RoboDK station: kr30 cnc 070119 curve 7 axis test 3.rdk

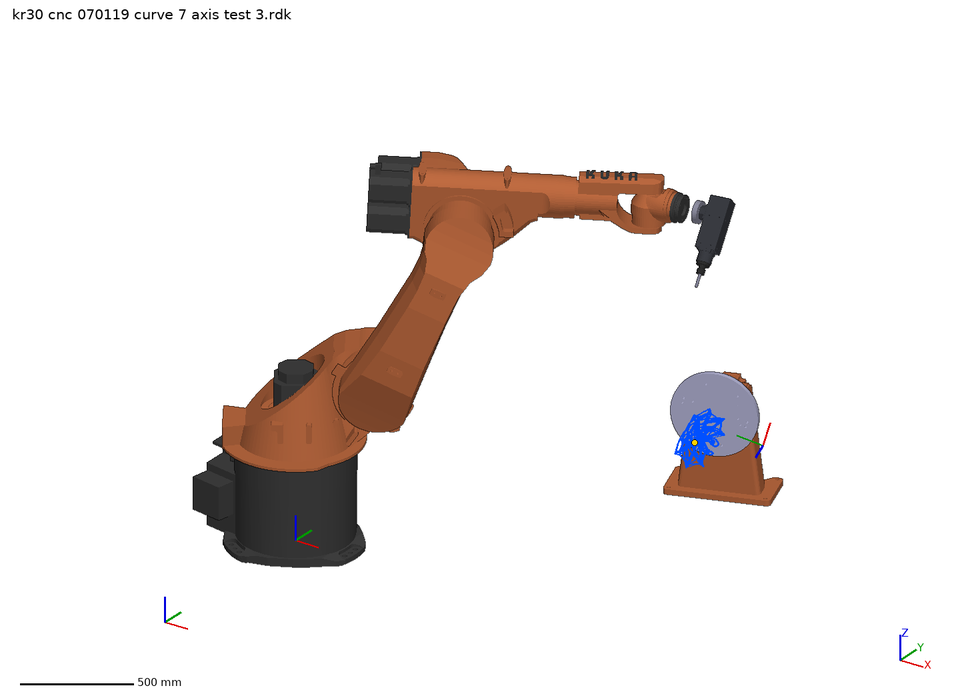
[picture v0: the station drawn from its stored meshes, robots at their saved joint values, targets as dots, program paths as lines]
Station kr30 cnc 070119 curve 7 axis test 3. Poses are relative to the parent item; angles as X-Y-Z fixed-axis rotations.
  - machining project Curve settings: C:/Temp/temp3/RhinoProject.stl | rotZ(0) | rotX(0)*rotY(0) | rotz(0) | onStart | onPathStart | onApproach | onPoint | onRetract | onFinish | onPathFinish | M_RunCode(%1)
  - frame KUKA KP1 MD250 Base at (0, 1000, 0) mm
    - robot KUKA KP1 MD250: 1 axes, payload 250 kg
        modified DH rows (alpha deg, a mm, theta deg, d mm): 0, 0, 0, 0
        base shift (1750, 1710, 820) mm, rotated rx 0 ry 90 rz -70 deg
        joint limits [-3600] to [3600]; home [0]; saved at [883.939]
      - frame Reference Rhino at (0, -260, 100) mm
        - object RhinoPart at (0, 0, 0) mm
  - frame KUKA KR 30 HA Base at (0, 2000, 0) mm
    - robot KUKA KR 30 HA: 6 axes, payload 30 kg, reach 2033 mm, repeatability 0.05 mm, weight 665 kg
        modified DH rows (alpha deg, a mm, theta deg, d mm): 0, 0, 0, 815; -90, 350, 0, 0; 0, 850, -90, 0; -90, 145, 0, 820; 90, 0, 0, 0; -90, 0, 180, 170
        joint limits [-185, -135, -120, -350, -119, -350] to [185, 35, 158, 350, 119, 350]; home [0, -90, 90, 0, 0, 0]; saved at [-33.388, -63.686, 66.526, 94.328, 22.372, -52.483]
      - tool 1/2" End Mill TCP, TCP at (337.71, -2.2, 160.57) mm, rotated rx 0 ry 90 rz 0 deg, size 415.8 x 102 x 153.6 mm
  - machining project RhinoPart Settings: rotZ(0) | rotX(0)*rotY(-65) | rotz(50) | onStart | onPathStart | onApproach | onPoint | onRetract | onFinish | onPathFinish | M_RunCode(%1)
  - program RhinoPart (1342 instructions, listed below)
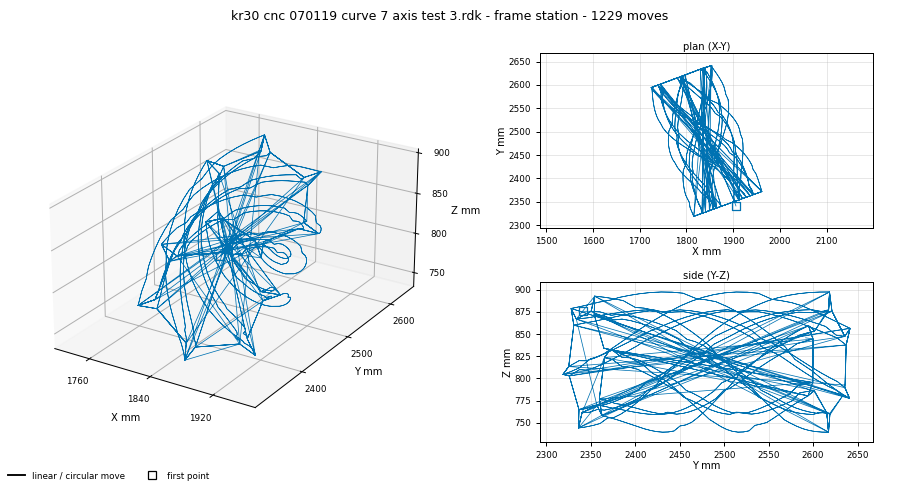
[picture p0: tool path of kr30 cnc 070119 curve 7 axis test 3.rdk in frame station, 1229 of 1229 moves have a stored position in this frame; points joined in program order, loops and branches not executed]

--- program RhinoPart (robot KUKA KR 30 HA) ---
  Set Ref.: Reference Rhino
  Set Tool: 1/2" End Mill TCP
  Show 1/2" End Mill TCP
  Set speed (1000.0 mm/s)
  MoveJ 1 to (58.93, 255.88, 300) mm, rotated rx 180 ry -65 rz 136 deg; joints [2.666, 0.348, 23.749, -54.366, 106.166, -75.82, 24.002]
  MoveL 2 to (58.93, 255.88, 300) mm, rotated rx 180 ry -65 rz 136 deg; joints [2.666, 0.348, 23.749, -54.366, 106.166, -75.82, 24.002]
  MoveL 3 to (58.93, 255.88, 290) mm, rotated rx 180 ry -65 rz 136 deg; joints [2.402, -0.635, 25.77, -54.277, 105.366, -75.09, 24.002]
  MoveL 4 to (58.93, 255.88, 290) mm, rotated rx 180 ry -65 rz 136 deg; joints [2.402, -0.635, 25.77, -54.277, 105.366, -75.09, 24.002]
  Set speed (60.0 mm/s)
  MoveL 5 to (37.11, 300.24, 290) mm, rotated rx -180 ry -65 rz -172.69 deg; joints [2.418, -1.215, 26.671, -54.196, 105.19, -74.811, -27.315]
  MoveL 6 to (-37.11, 208.63, 290) mm, rotated rx -180 ry -65 rz 14.16 deg; joints [2.386, -0.033, 24.818, -54.365, 105.558, -75.393, 145.844]
  Set speed (60.0 mm/s)
  MoveL 7 to (-58.93, 252.99, 290) mm, rotated rx -180 ry -65 rz -33.22 deg; joints [2.401, -0.598, 25.711, -54.282, 105.378, -75.109, 193.216]
  MoveL 8 to (21.11, 199.39, 290) mm, rotated rx -180 ry -65 rz 69.21 deg; joints [2.383, 0.084, 24.632, -54.382, 105.596, -75.453, 90.794]
  Set speed (60.0 mm/s)
  MoveL 9 to (34.79, 183.72, 290) mm, rotated rx -180 ry -65 rz 74.51 deg; joints [2.31, 3.521, 18.897, -54.969, 106.871, -77.447, 85.485]
  MoveL 10 to (21.11, 199.39, 290) mm, rotated rx -180 ry -65 rz 69.21 deg; joints [2.383, 0.084, 24.632, -54.382, 105.596, -75.453, 90.794]
  Set speed (60.0 mm/s)
  MoveL 11 to (-28.22, 202.67, 290) mm, rotated rx 180 ry -65 rz 23.79 deg; joints [2.384, 0.043, 24.698, -54.376, 105.583, -75.432, 136.207]
  MoveL 12 to (-43.85, 188.95, 290) mm, rotated rx 180 ry -65 rz 18.32 deg; joints [2.311, 3.444, 19.031, -54.954, 106.839, -77.397, 141.679]
  Set speed (60.0 mm/s)
  MoveL 13 to (-28.22, 202.67, 290) mm, rotated rx -180 ry -65 rz 23.79 deg; joints [2.384, 0.043, 24.698, -54.376, 105.583, -75.432, 136.207]
  MoveL 14 to (-43.85, 188.95, 290) mm, rotated rx 180 ry -65 rz 18.32 deg; joints [2.311, 3.444, 19.031, -54.954, 106.839, -77.397, 141.679]
  Set speed (60.0 mm/s)
  MoveL 15 to (-37.11, 208.63, 290) mm, rotated rx -180 ry -65 rz 14.16 deg; joints [2.386, -0.033, 24.818, -54.365, 105.558, -75.393, 145.844]
  MoveL 16 to (-78.63, 259.66, 290) mm, rotated rx 180 ry -65 rz -39.75 deg; joints [2.329, 2.455, 20.731, -54.77, 106.443, -76.78, 199.755]
  Set speed (60.0 mm/s)
  MoveL 17 to (-58.93, 252.99, 290) mm, rotated rx -180 ry -65 rz -33.22 deg; joints [2.401, -0.598, 25.711, -54.282, 105.378, -75.109, 193.216]
  MoveL 18 to (-78.63, 259.66, 290) mm, rotated rx -180 ry -65 rz -39.75 deg; joints [2.329, 2.455, 20.731, -54.77, 106.443, -76.78, 199.755]
  Set speed (60.0 mm/s)
  MoveL 19 to (-58.22, 263.67, 290) mm, rotated rx -180 ry -65 rz -43.61 deg; joints [2.405, -0.736, 25.927, -54.263, 105.335, -75.041, 203.606]
  MoveL 20 to (-30.72, 304.75, 290) mm, rotated rx -180 ry -65 rz -95.53 deg; joints [2.42, -1.275, 26.764, -54.188, 105.172, -74.782, 255.533]
  Set speed (60.0 mm/s)
  MoveL 21 to (-58.22, 263.67, 290) mm, rotated rx -180 ry -65 rz -43.61 deg; joints [2.405, -0.736, 25.927, -54.263, 105.335, -75.041, 203.606]
  MoveL 22 to (-30.72, 304.75, 290) mm, rotated rx -180 ry -65 rz -95.53 deg; joints [2.42, -1.275, 26.764, -54.188, 105.172, -74.782, 255.533]
  Set speed (60.0 mm/s)
  MoveL 23 to (-34.79, 325.15, 290) mm, rotated rx 180 ry -65 rz -101.9 deg; joints [2.347, 1.599, 22.168, -54.622, 106.121, -76.277, 261.899]
  MoveL 24 to (-21.11, 309.47, 290) mm, rotated rx -180 ry -65 rz -106.89 deg; joints [2.421, -1.338, 26.861, -54.18, 105.153, -74.752, 266.89]
  Set speed (60.0 mm/s)
  MoveL 25 to (-34.79, 325.15, 290) mm, rotated rx -180 ry -65 rz -101.9 deg; joints [2.347, 1.599, 22.168, -54.622, 106.121, -76.277, 261.899]
  MoveL 26 to (-21.11, 309.47, 290) mm, rotated rx -180 ry -65 rz -106.89 deg; joints [2.421, -1.338, 26.861, -54.18, 105.153, -74.752, 266.89]
  Set speed (60.0 mm/s)
  MoveL 27 to (28.22, 306.19, 290) mm, rotated rx 180 ry -65 rz -161.42 deg; joints [2.42, -1.294, 26.794, -54.186, 105.166, -74.773, 321.418]
  MoveL 28 to (43.85, 319.91, 290) mm, rotated rx -180 ry -65 rz -166.2 deg; joints [2.345, 1.666, 22.057, -54.633, 106.146, -76.315, 326.197]
  Set speed (60.0 mm/s)
  MoveL 29 to (28.22, 306.19, 290) mm, rotated rx -180 ry -65 rz -161.42 deg; joints [2.42, -1.294, 26.794, -54.186, 105.166, -74.773, 321.418]
  MoveL 30 to (43.85, 319.91, 290) mm, rotated rx -180 ry -65 rz -166.2 deg; joints [2.345, 1.666, 22.057, -54.633, 106.146, -76.315, 326.197]
  Set speed (60.0 mm/s)
  MoveL 31 to (37.11, 300.24, 290) mm, rotated rx -180 ry -65 rz -172.69 deg; joints [2.418, -1.215, 26.671, -54.196, 105.19, -74.811, 332.685]
  MoveL 32 to (78.63, 249.2, 290) mm, rotated rx 180 ry -65 rz 132.18 deg; joints [2.326, 2.596, 20.491, -54.795, 106.498, -76.866, 387.819]
  Set speed (60.0 mm/s)
  MoveL 33 to (58.93, 255.88, 290) mm, rotated rx -180 ry -65 rz 136 deg; joints [2.402, -0.635, 25.77, -54.277, 105.366, -75.09, 384.002]
  MoveL 34 to (78.63, 249.2, 290) mm, rotated rx 180 ry -65 rz 132.18 deg; joints [2.326, 2.596, 20.491, -54.795, 106.498, -76.866, 387.819]
  Set speed (60.0 mm/s)
  MoveL 35 to (58.22, 245.2, 290) mm, rotated rx -180 ry -65 rz 125.73 deg; joints [2.398, -0.498, 25.554, -54.297, 105.409, -75.158, 394.265]
  MoveL 36 to (30.72, 204.12, 290) mm, rotated rx -180 ry -65 rz 78.8 deg; joints [2.384, 0.024, 24.728, -54.373, 105.577, -75.423, 441.204]
  Set speed (60.0 mm/s)
  MoveL 37 to (58.22, 245.2, 290) mm, rotated rx -180 ry -65 rz 125.73 deg; joints [2.398, -0.498, 25.554, -54.297, 105.409, -75.158, 394.265]
  MoveL 38 to (30.72, 204.12, 290) mm, rotated rx -180 ry -65 rz 78.8 deg; joints [2.384, 0.024, 24.728, -54.373, 105.577, -75.423, 441.204]
  Set speed (60.0 mm/s)
  MoveL 39 to (34.79, 183.72, 290) mm, rotated rx 180 ry -65 rz 74.51 deg; joints [2.31, 3.521, 18.897, -54.969, 106.871, -77.447, 445.485]
  MoveL 40 to (-36.94, 300.02, -0.17) mm, rotated rx -180 ry -65 rz -46.62 deg; joints [-6.447, 6.894, 10.028, -66.341, 87.316, -50.83, 606.623]
  Set speed (60.0 mm/s)
  MoveL 41 to (10.28, 312.41, -0.04) mm, rotated rx -180 ry -65 rz -100.95 deg; joints [-6.444, 6.854, 10.028, -66.338, 87.334, -50.865, 660.953]
  MoveL 42 to (-36.94, 300.02, -0.17) mm, rotated rx -180 ry -65 rz -46.62 deg; joints [-6.447, 6.894, 10.028, -66.341, 87.316, -50.83, 606.623]
  Set speed (60.0 mm/s)
  MoveL 43 to (-55.59, 310.29, 0) mm, rotated rx -180 ry -65 rz -52.13 deg; joints [-6.306, 15.735, -5.818, -64.17, 93.982, -66.18, 602.13]
  MoveL 44 to (-44.28, 292.75, -0.25) mm, rotated rx -180 ry -65 rz -35.52 deg; joints [-6.449, 6.917, 10.028, -66.342, 87.305, -50.809, 595.516]
  Set speed (60.0 mm/s)
  MoveL 45 to (-55.59, 310.29, 0) mm, rotated rx -180 ry -65 rz -52.13 deg; joints [-6.306, 0.053, 25.874, -64.052, 86.954, -51.786, 602.13]
  MoveL 46 to (-44.28, 292.75, -0.25) mm, rotated rx -180 ry -65 rz -35.52 deg; joints [-6.449, 6.917, 10.028, -66.342, 87.305, -50.809, 595.516]
  Set speed (60.0 mm/s)
  MoveL 47 to (-57.47, 247.5, -0.72) mm, rotated rx -180 ry -65 rz 14.89 deg; joints [-6.459, 7.056, 10.028, -66.351, 87.24, -50.686, 545.106]
  MoveL 48 to (-76.17, 234.21, 0) mm, rotated rx 180 ry -65 rz 8.7 deg; joints [-6.319, 15.262, -4.528, -64.124, 93.614, -65.448, 541.297]
  Set speed (60.0 mm/s)
  MoveL 49 to (-57.47, 247.5, -0.72) mm, rotated rx 180 ry -65 rz 14.89 deg; joints [-6.459, 7.056, 10.028, -66.351, 87.24, -50.686, 545.106]
  MoveL 50 to (-76.17, 234.21, 0) mm, rotated rx 180 ry -65 rz 8.7 deg; joints [-6.319, 15.262, -4.528, -64.124, 93.614, -65.448, 541.297]
  Set speed (60.0 mm/s)
  MoveL 51 to (-55.23, 237.63, -0.82) mm, rotated rx -180 ry -65 rz 24.99 deg; joints [-6.461, 7.085, 10.028, -66.353, 87.227, -50.66, 535.014]
  MoveL 52 to (-23.82, 202.61, -1.14) mm, rotated rx 180 ry -65 rz 71.39 deg; joints [-6.468, 7.179, 10.028, -66.359, 87.183, -50.576, 488.615]
  Set speed (60.0 mm/s)
  MoveL 53 to (-55.23, 237.63, -0.82) mm, rotated rx -180 ry -65 rz 24.99 deg; joints [-6.461, 7.085, 10.028, -66.353, 87.227, -50.66, 535.014]
  MoveL 54 to (-23.82, 202.61, -1.14) mm, rotated rx 180 ry -65 rz 71.39 deg; joints [-6.468, 7.179, 10.028, -66.359, 87.183, -50.576, 488.615]
  Set speed (60.0 mm/s)
  MoveL 55 to (-20.57, 178.36, 0) mm, rotated rx 180 ry -65 rz 65.86 deg; joints [-6.327, 14.897, -3.558, -64.093, 93.342, -64.907, 484.144]
  MoveL 56 to (-14.1, 199.28, -1.17) mm, rotated rx -180 ry -65 rz 80.93 deg; joints [-6.469, 7.186, 10.028, -66.36, 87.179, -50.57, 479.071]
  Set speed (60.0 mm/s)
  MoveL 57 to (-20.57, 178.36, 0) mm, rotated rx -180 ry -65 rz 65.86 deg; joints [-6.327, 1.451, 23.614, -64.022, 87.314, -52.57, 484.144]
  MoveL 58 to (-14.1, 199.28, -1.17) mm, rotated rx -180 ry -65 rz 80.93 deg; joints [-6.469, 7.186, 10.028, -66.36, 87.179, -50.57, 479.071]
  Set speed (60.0 mm/s)
  MoveL 59 to (33.26, 208.35, -1.05) mm, rotated rx -180 ry -65 rz 126.44 deg; joints [-6.466, 7.153, 10.028, -66.357, 87.195, -50.6, 433.558]
  MoveL 60 to (55.59, 198.58, 0) mm, rotated rx -180 ry -65 rz 122.15 deg; joints [-6.324, 15.031, -3.912, -64.104, 93.441, -65.104, 427.85]
  Set speed (60.0 mm/s)
  MoveL 61 to (33.26, 208.35, -1.05) mm, rotated rx 180 ry -65 rz 126.44 deg; joints [-6.466, 7.153, 10.028, -66.357, 87.195, -50.6, 433.558]
  MoveL 62 to (55.59, 198.58, 0) mm, rotated rx -180 ry -65 rz 122.15 deg; joints [-6.324, 15.031, -3.912, -64.104, 93.441, -65.104, 427.85]
  Set speed (60.0 mm/s)
  MoveL 63 to (41.3, 215.27, -0.99) mm, rotated rx -180 ry -65 rz 136.17 deg; joints [-6.465, 7.133, 10.028, -66.356, 87.204, -50.617, 423.831]
  MoveL 64 to (57.25, 262.28, -0.53) mm, rotated rx 180 ry -65 rz -175.75 deg; joints [-6.455, 7, 10.028, -66.348, 87.266, -50.736, 375.746]
  Set speed (60.0 mm/s)
  MoveL 65 to (41.3, 215.27, -0.99) mm, rotated rx -180 ry -65 rz 136.17 deg; joints [-6.465, 7.133, 10.028, -66.356, 87.204, -50.617, 423.831]
  MoveL 66 to (57.25, 262.28, -0.53) mm, rotated rx 180 ry -65 rz -175.75 deg; joints [-6.455, 7, 10.028, -66.348, 87.266, -50.736, 375.746]
  Set speed (60.0 mm/s)
  MoveL 67 to (76.17, 274.65, 0) mm, rotated rx 180 ry -65 rz -179.11 deg; joints [-6.312, 0.429, 25.273, -64.043, 87.048, -51.99, 369.111]
  MoveL 68 to (54.99, 272.92, -0.43) mm, rotated rx -180 ry -65 rz -165.16 deg; joints [-6.453, 6.969, 10.028, -66.346, 87.28, -50.763, 365.162]
  Set speed (60.0 mm/s)
  MoveL 69 to (76.17, 274.65, 0) mm, rotated rx 180 ry -65 rz -179.11 deg; joints [-6.312, 15.517, -5.217, -64.148, 93.809, -65.837, 369.111]
  MoveL 70 to (54.99, 272.92, -0.43) mm, rotated rx -180 ry -65 rz -165.16 deg; joints [-6.453, 6.969, 10.028, -66.346, 87.28, -50.763, 365.162]
  Set speed (60.0 mm/s)
  MoveL 71 to (20.67, 309.5, -0.07) mm, rotated rx 180 ry -65 rz -112.4 deg; joints [-6.445, 6.863, 10.028, -66.339, 87.33, -50.857, 312.405]
  MoveL 72 to (20.57, 330.51, 0) mm, rotated rx 180 ry -65 rz -116.27 deg; joints [-6.302, -0.161, 26.213, -64.056, 86.902, -51.671, 306.267]
  Set speed (60.0 mm/s)
  MoveL 73 to (20.67, 309.5, -0.07) mm, rotated rx 180 ry -65 rz -112.4 deg; joints [-6.445, 6.863, 10.028, -66.339, 87.33, -50.857, 312.405]
  MoveL 74 to (20.57, 330.51, 0) mm, rotated rx -180 ry -65 rz -116.27 deg; joints [-6.302, 15.857, -6.157, -64.183, 94.08, -66.375, 306.267]
  Set speed (60.0 mm/s)
  MoveL 75 to (10.28, 312.41, -0.04) mm, rotated rx -180 ry -65 rz -100.95 deg; joints [-6.444, 6.854, 10.028, -66.338, 87.334, -50.865, 300.953]
  MoveL 76 to (-36.94, 300.02, -0.17) mm, rotated rx -180 ry -65 rz -46.62 deg; joints [-6.447, 6.894, 10.028, -66.341, 87.316, -50.83, 246.623]
  Set speed (60.0 mm/s)
  MoveL 77 to (-37.93, 298.04, 9.24) mm, rotated rx -180 ry -65 rz -42.11 deg; joints [-6.172, 6.893, 10.028, -66.266, 87.557, -50.725, 242.114]
  MoveL 78 to (-39.11, 295.92, 18.61) mm, rotated rx 180 ry -65 rz -37.19 deg; joints [-5.899, 6.893, 10.028, -66.19, 87.796, -50.619, 237.19]
  MoveL 79 to (-47.39, 289.5, 30) mm, rotated rx 180 ry -65 rz -41.9 deg; joints [-5.427, 15.454, -6.498, -64.065, 95.181, -66.668, 231.9]
  MoveL 80 to (-50.45, 284.92, 40) mm, rotated rx 180 ry -65 rz -36.29 deg; joints [-5.152, 14.792, -5.154, -63.954, 95.127, -65.933, 226.29]
  MoveL 81 to (-53.21, 279.8, 50) mm, rotated rx -180 ry -65 rz -30.41 deg; joints [-4.877, 14.047, -3.641, -63.835, 95.031, -65.12, 220.409]
  MoveL 82 to (-55.55, 274.16, 60) mm, rotated rx -180 ry -65 rz -24.3 deg; joints [-4.603, 13.189, -1.895, -63.704, 94.88, -64.202, 214.303]
  MoveL 83 to (-57.35, 268.08, 70) mm, rotated rx -180 ry -65 rz -18.01 deg; joints [-4.33, 12.157, 0.203, -63.558, 94.646, -63.125, 208.015]
  MoveL 84 to (-58.51, 261.62, 80) mm, rotated rx -180 ry -65 rz -11.59 deg; joints [-4.058, 10.802, 2.956, -63.39, 94.259, -61.752, 201.589]
  MoveL 85 to (-58.95, 254.91, 90) mm, rotated rx -180 ry -65 rz -5.06 deg; joints [-3.787, 8.124, 8.381, -63.151, 93.257, -59.174, 195.064]
  MoveL 86 to (-57.83, 250.73, 99.18) mm, rotated rx -180 ry -65 rz 1.52 deg; joints [-3.517, 7.316, 10.028, -63.024, 93.108, -58.308, 188.479]
  MoveL 87 to (-56.49, 246.88, 108.28) mm, rotated rx -180 ry -65 rz 8.13 deg; joints [-3.247, 7.323, 10.028, -62.936, 93.334, -58.185, 181.868]
  MoveL 88 to (-55.46, 234.45, 120) mm, rotated rx 180 ry -65 rz 4.74 deg; joints [-2.737, 15.802, -6.649, -62.008, 101.438, -74.132, 175.264]
  MoveL 89 to (-52.68, 227.97, 130) mm, rotated rx 180 ry -65 rz 11.3 deg; joints [-2.465, 15.019, -5.058, -61.795, 101.294, -73.276, 168.698]
  MoveL 90 to (-49.15, 221.88, 140) mm, rotated rx -180 ry -65 rz 17.8 deg; joints [-2.195, 14.134, -3.264, -61.562, 101.096, -72.332, 162.199]
  MoveL 91 to (-44.94, 216.28, 150) mm, rotated rx 180 ry -65 rz 24.21 deg; joints [-1.925, 13.101, -1.172, -61.304, 100.823, -71.256, 155.793]
  MoveL 92 to (-40.17, 211.29, 160) mm, rotated rx 180 ry -65 rz 30.49 deg; joints [-1.655, 11.813, 1.429, -61.006, 100.419, -69.957, 149.508]
  MoveL 93 to (-34.94, 206.95, 170) mm, rotated rx 180 ry -65 rz 36.63 deg; joints [-1.387, 9.888, 5.314, -60.614, 99.691, -68.09, 143.368]
  MoveL 94 to (-30.4, 204.81, 179.39) mm, rotated rx 180 ry -65 rz 42.6 deg; joints [-1.119, 7.55, 10.028, -60.183, 98.74, -65.868, 137.399]
  MoveL 95 to (-26.84, 204.2, 188.29) mm, rotated rx -180 ry -65 rz 48.37 deg; joints [-0.852, 7.543, 10.028, -60.083, 98.964, -65.746, 131.627]
  MoveL 96 to (-17.8, 198.23, 200) mm, rotated rx 180 ry -65 rz 43.92 deg; joints [-0.31, 16.045, -7.071, -60.462, 107.755, -81.941, 126.077]
  MoveL 97 to (-12.04, 196.73, 210) mm, rotated rx -180 ry -65 rz 49.22 deg; joints [-0.041, 15.22, -5.426, -60.15, 107.58, -81.056, 120.776]
  MoveL 98 to (-6.46, 195.84, 220) mm, rotated rx 180 ry -65 rz 54.25 deg; joints [0.227, 14.29, -3.573, -59.809, 107.346, -80.08, 115.751]
  MoveL 99 to (-1.16, 195.49, 230) mm, rotated rx 180 ry -65 rz 58.97 deg; joints [0.494, 13.205, -1.411, -59.428, 107.028, -78.968, 111.029]
  MoveL 100 to (3.78, 195.6, 240) mm, rotated rx -180 ry -65 rz 63.36 deg; joints [0.761, 11.852, 1.291, -58.981, 106.561, -77.618, 106.641]
  MoveL 101 to (8.28, 196.07, 250) mm, rotated rx 180 ry -65 rz 67.38 deg; joints [1.027, 9.8, 5.404, -58.368, 105.709, -75.646, 102.617]
  MoveL 102 to (10.36, 197.38, 259.21) mm, rotated rx -180 ry -65 rz 71.01 deg; joints [1.292, 7.494, 10.028, -57.722, 104.698, -73.469, 98.987]
  MoveL 103 to (10.58, 198.92, 267.9) mm, rotated rx -180 ry -65 rz 74.21 deg; joints [1.556, 7.475, 10.028, -57.611, 104.921, -73.346, 95.785]
  MoveL 104 to (18.74, 198.54, 280) mm, rotated rx -180 ry -65 rz 66.96 deg; joints [2.118, -0.825, 26.508, -54.319, 104.838, -74.784, 93.043]
  MoveL 105 to (21.11, 199.39, 290) mm, rotated rx -180 ry -65 rz 69.21 deg; joints [2.383, 0.084, 24.632, -54.382, 105.596, -75.453, 90.794]
  MoveL 106 to (10.16, 312.5, 0) mm, rotated rx -180 ry -65 rz -110.95 deg; joints [-6.256, -2.705, 30.12, -64.109, 86.344, -50.426, -59.047]
  Set speed (60.0 mm/s)
  MoveL 107 to (-36.94, 300.02, -0.17) mm, rotated rx -180 ry -65 rz -46.62 deg; joints [-6.447, 6.894, 10.028, -66.341, 87.316, -50.83, -113.377]
  MoveL 108 to (-28.22, 202.67, 290) mm, rotated rx -180 ry -65 rz 23.79 deg; joints [2.384, 14.562, -4.643, -58.828, 113.78, -88.566, -223.793]
  Set speed (60.0 mm/s)
  MoveL 109 to (21.11, 199.39, 290) mm, rotated rx 180 ry -65 rz 69.21 deg; joints [2.383, 14.538, -4.577, -58.812, 113.757, -88.527, -269.206]
  MoveL 110 to (-28.22, 202.67, 290) mm, rotated rx 180 ry -65 rz 23.79 deg; joints [2.384, 14.562, -4.643, -58.828, 113.78, -88.566, -223.793]
  Set speed (60.0 mm/s)
  MoveL 111 to (-30.4, 203.93, 280) mm, rotated rx -180 ry -65 rz 21.53 deg; joints [2.12, 15.518, -6.548, -59.292, 114.044, -89.604, -221.533]
  MoveL 112 to (-35.6, 209.96, 268.01) mm, rotated rx -180 ry -65 rz 28.77 deg; joints [1.558, 7.454, 10.028, -57.615, 104.934, -73.363, -218.768]
  MoveL 113 to (-36.68, 209.15, 259.36) mm, rotated rx -180 ry -65 rz 25.53 deg; joints [1.295, 7.465, 10.028, -57.727, 104.716, -73.493, -215.528]
  MoveL 114 to (-39.07, 210.28, 250) mm, rotated rx -180 ry -65 rz 21.84 deg; joints [1.031, 10.179, 4.562, -58.478, 105.955, -76.054, -211.841]
  MoveL 115 to (-42.34, 213.41, 240) mm, rotated rx -180 ry -65 rz 17.73 deg; joints [0.766, 12.098, 0.7, -59.067, 106.743, -77.925, -207.735]
  MoveL 116 to (-45.62, 217.1, 230) mm, rotated rx 180 ry -65 rz 13.24 deg; joints [0.501, 13.423, -1.967, -59.516, 107.205, -79.27, -203.236]
  MoveL 117 to (-48.8, 221.36, 220) mm, rotated rx 180 ry -65 rz 8.37 deg; joints [0.235, 14.498, -4.131, -59.902, 107.529, -80.393, -198.371]
  MoveL 118 to (-51.74, 226.19, 210) mm, rotated rx 180 ry -65 rz 3.16 deg; joints [-0.032, 15.423, -5.997, -60.249, 107.77, -81.387, -193.164]
  MoveL 119 to (-54.33, 231.55, 200) mm, rotated rx 180 ry -65 rz -2.36 deg; joints [-0.3, 16.246, -7.66, -60.568, 107.955, -82.291, -187.64]
  MoveL 120 to (-56.06, 240.96, 188.77) mm, rotated rx 180 ry -65 rz 1.82 deg; joints [-0.842, 7.444, 10.028, -60.093, 99.023, -65.828, -181.825]
  MoveL 121 to (-57.9, 243.94, 179.9) mm, rotated rx 180 ry -65 rz -4.26 deg; joints [-1.108, 7.441, 10.028, -60.193, 98.804, -65.959, -175.742]
  MoveL 122 to (-58.8, 250.25, 170) mm, rotated rx -180 ry -65 rz -10.58 deg; joints [-1.375, 3.96, 17.054, -59.877, 96.815, -62.987, -169.418]
  MoveL 123 to (-58.89, 257.04, 160) mm, rotated rx -180 ry -65 rz -17.12 deg; joints [-1.643, 2.411, 20.173, -59.84, 95.811, -61.746, -162.877]
  MoveL 124 to (-58.18, 263.92, 150) mm, rotated rx -180 ry -65 rz -23.85 deg; joints [-1.911, 1.246, 22.515, -59.862, 95.006, -60.848, -156.149]
  MoveL 125 to (-56.65, 270.74, 140) mm, rotated rx 180 ry -65 rz -30.74 deg; joints [-2.181, 0.277, 24.46, -59.914, 94.304, -60.125, -149.263]
  MoveL 126 to (-54.3, 277.38, 130) mm, rotated rx 180 ry -65 rz -37.75 deg; joints [-2.452, -0.566, 26.151, -59.986, 93.667, -59.512, -142.251]
  MoveL 127 to (-51.17, 283.7, 120) mm, rotated rx -180 ry -65 rz -44.85 deg; joints [-2.723, -1.316, 27.656, -60.073, 93.079, -58.979, -135.149]
  MoveL 128 to (-44.05, 291.51, 108.86) mm, rotated rx -180 ry -65 rz -42.01 deg; joints [-3.234, 7.183, 10.028, -62.94, 93.409, -58.304, -127.994]
  MoveL 129 to (-42.07, 295.25, 99.75) mm, rotated rx -180 ry -65 rz -49.17 deg; joints [-3.504, 7.179, 10.028, -63.026, 93.181, -58.425, -120.828]
  MoveL 130 to (-37.86, 299.62, 90) mm, rotated rx -180 ry -65 rz -56.3 deg; joints [-3.775, 4.333, 15.773, -63.009, 91.636, -55.955, -113.695]
  MoveL 131 to (-32.46, 303.64, 80) mm, rotated rx 180 ry -65 rz -63.36 deg; joints [-4.047, 2.783, 18.905, -63.08, 90.693, -54.661, -106.643]
  MoveL 132 to (-26.8, 306.94, 70) mm, rotated rx -180 ry -65 rz -70.28 deg; joints [-4.32, 1.68, 21.137, -63.178, 89.957, -53.768, -99.72]
  MoveL 133 to (-21, 309.52, 60) mm, rotated rx -180 ry -65 rz -77.02 deg; joints [-4.594, 0.789, 22.944, -63.291, 89.32, -53.063, -92.977]
  MoveL 134 to (-15.19, 311.39, 50) mm, rotated rx 180 ry -65 rz -83.54 deg; joints [-4.869, 0.031, 24.487, -63.413, 88.743, -52.474, -86.464]
  MoveL 135 to (-9.5, 312.61, 40) mm, rotated rx 180 ry -65 rz -89.77 deg; joints [-5.145, -0.633, 25.843, -63.543, 88.21, -51.966, -80.231]
  MoveL 136 to (-4.03, 313.25, 30) mm, rotated rx -180 ry -65 rz -95.67 deg; joints [-5.421, -1.225, 27.059, -63.678, 87.71, -51.518, -74.327]
  MoveL 137 to (5.28, 311.14, 18.82) mm, rotated rx 180 ry -65 rz -91.2 deg; joints [-5.894, 6.832, 10.028, -66.187, 87.825, -50.673, -68.799]
  MoveL 138 to (7.88, 311.77, 9.41) mm, rotated rx -180 ry -65 rz -96.31 deg; joints [-6.169, 6.842, 10.028, -66.263, 87.58, -50.77, -63.692]
  MoveL 139 to (10.28, 312.41, -0.04) mm, rotated rx -180 ry -65 rz -100.95 deg; joints [-6.444, 6.854, 10.028, -66.338, 87.334, -50.865, -59.047]
  MoveL 140 to (-36.94, 300.02, -0.17) mm, rotated rx -180 ry -65 rz -46.62 deg; joints [-6.447, 6.894, 10.028, -66.341, 87.316, -50.83, -113.377]
  Set speed (60.0 mm/s)
  MoveL 141 to (-37.93, 298.04, 9.24) mm, rotated rx -180 ry -65 rz -42.11 deg; joints [-6.172, 6.893, 10.028, -66.266, 87.557, -50.725, -117.886]
  MoveL 142 to (-39.11, 295.92, 18.61) mm, rotated rx -180 ry -65 rz -37.19 deg; joints [-5.899, 6.893, 10.028, -66.19, 87.796, -50.619, -122.81]
  MoveL 143 to (-47.39, 289.5, 30) mm, rotated rx -180 ry -65 rz -41.9 deg; joints [-5.427, 15.454, -6.498, -64.065, 95.181, -66.668, -128.1]
  MoveL 144 to (-50.45, 284.92, 40) mm, rotated rx -180 ry -65 rz -36.29 deg; joints [-5.152, 14.792, -5.154, -63.954, 95.127, -65.933, -133.71]
  MoveL 145 to (-53.21, 279.8, 50) mm, rotated rx 180 ry -65 rz -30.41 deg; joints [-4.877, 14.047, -3.641, -63.835, 95.031, -65.12, -139.591]
  MoveL 146 to (-55.55, 274.16, 60) mm, rotated rx -180 ry -65 rz -24.3 deg; joints [-4.603, 13.189, -1.895, -63.704, 94.88, -64.202, -145.697]
  MoveL 147 to (-57.35, 268.08, 70) mm, rotated rx -180 ry -65 rz -18.01 deg; joints [-4.33, 12.157, 0.203, -63.558, 94.646, -63.125, -151.985]
  MoveL 148 to (-58.51, 261.62, 80) mm, rotated rx -180 ry -65 rz -11.59 deg; joints [-4.058, 10.802, 2.956, -63.39, 94.259, -61.752, -158.411]
  MoveL 149 to (-58.95, 254.91, 90) mm, rotated rx -180 ry -65 rz -5.06 deg; joints [-3.787, 8.124, 8.381, -63.151, 93.257, -59.174, -164.936]
  MoveL 150 to (-57.83, 250.73, 99.18) mm, rotated rx 180 ry -65 rz 1.52 deg; joints [-3.517, 7.316, 10.028, -63.024, 93.108, -58.308, -171.521]
  MoveL 151 to (-56.49, 246.88, 108.28) mm, rotated rx -180 ry -65 rz 8.13 deg; joints [-3.247, 7.323, 10.028, -62.936, 93.334, -58.185, -178.132]
  MoveL 152 to (-55.46, 234.45, 120) mm, rotated rx 180 ry -65 rz 4.74 deg; joints [-2.737, 15.802, -6.649, -62.008, 101.438, -74.132, -184.736]
  MoveL 153 to (-52.68, 227.97, 130) mm, rotated rx -180 ry -65 rz 11.3 deg; joints [-2.465, 15.019, -5.058, -61.795, 101.294, -73.276, -191.302]
  MoveL 154 to (-49.15, 221.88, 140) mm, rotated rx -180 ry -65 rz 17.8 deg; joints [-2.195, 14.134, -3.264, -61.562, 101.096, -72.332, -197.801]
  MoveL 155 to (-44.94, 216.28, 150) mm, rotated rx -180 ry -65 rz 24.21 deg; joints [-1.925, 13.101, -1.172, -61.304, 100.823, -71.256, -204.207]
  MoveL 156 to (-40.17, 211.29, 160) mm, rotated rx -180 ry -65 rz 30.49 deg; joints [-1.655, 11.813, 1.429, -61.006, 100.419, -69.957, -210.492]
  MoveL 157 to (-34.94, 206.95, 170) mm, rotated rx -180 ry -65 rz 36.63 deg; joints [-1.387, 9.888, 5.314, -60.614, 99.691, -68.09, -216.632]
  MoveL 158 to (-30.4, 204.81, 179.39) mm, rotated rx 180 ry -65 rz 42.6 deg; joints [-1.119, 7.55, 10.028, -60.183, 98.74, -65.868, -222.601]
  MoveL 159 to (-26.84, 204.2, 188.29) mm, rotated rx -180 ry -65 rz 48.37 deg; joints [-0.852, 7.543, 10.028, -60.083, 98.964, -65.746, -228.373]
  MoveL 160 to (-17.8, 198.23, 200) mm, rotated rx 180 ry -65 rz 43.92 deg; joints [-0.31, -0.877, 27.127, -56.961, 98.729, -66.788, -233.923]
  MoveL 161 to (-12.04, 196.73, 210) mm, rotated rx 180 ry -65 rz 49.22 deg; joints [-0.041, -0.074, 25.482, -56.935, 99.391, -67.369, -239.224]
  MoveL 162 to (-6.46, 195.84, 220) mm, rotated rx 180 ry -65 rz 54.25 deg; joints [0.227, 0.829, 23.629, -56.936, 100.113, -68.042, -244.249]
  MoveL 163 to (-1.16, 195.49, 230) mm, rotated rx -180 ry -65 rz 58.97 deg; joints [0.494, 1.884, 21.467, -56.975, 100.922, -68.85, -248.971]
  MoveL 164 to (3.78, 195.6, 240) mm, rotated rx -180 ry -65 rz 63.36 deg; joints [0.761, 3.206, 18.764, -57.079, 101.88, -69.896, -253.359]
  MoveL 165 to (8.28, 196.07, 250) mm, rotated rx 180 ry -65 rz 67.38 deg; joints [1.027, 5.224, 14.652, -57.347, 103.223, -71.562, -257.383]
  MoveL 166 to (10.36, 197.38, 259.21) mm, rotated rx -180 ry -65 rz 71.01 deg; joints [1.292, 7.494, 10.028, -57.722, 104.698, -73.469, -261.013]
  MoveL 167 to (10.58, 198.92, 267.9) mm, rotated rx -180 ry -65 rz 74.21 deg; joints [1.556, 7.475, 10.028, -57.611, 104.921, -73.346, -264.215]
  MoveL 168 to (18.74, 198.54, 280) mm, rotated rx -180 ry -65 rz 66.96 deg; joints [2.118, -0.825, 26.508, -54.319, 104.838, -74.784, -266.957]
  MoveL 169 to (21.11, 199.39, 290) mm, rotated rx -180 ry -65 rz 69.21 deg; joints [2.383, 0.084, 24.632, -54.382, 105.596, -75.453, -269.206]
  MoveL 170 to (34.79, 183.72, 290) mm, rotated rx 180 ry -65 rz 74.51 deg; joints [2.31, 3.521, 18.897, -54.969, 106.871, -77.447, -274.515]
  Set speed (60.0 mm/s)
  MoveL 171 to (21.11, 199.39, 290) mm, rotated rx 180 ry -65 rz 69.21 deg; joints [2.383, 0.084, 24.632, -54.382, 105.596, -75.453, -269.206]
  MoveL 172 to (-55.59, 310.29, 0) mm, rotated rx 180 ry -65 rz -52.13 deg; joints [-6.306, 0.053, 25.874, -64.052, 86.954, -51.786, -117.87]
  Set speed (60.0 mm/s)
  MoveL 173 to (-36.94, 300.02, -0.17) mm, rotated rx -180 ry -65 rz -46.62 deg; joints [-6.447, 6.894, 10.028, -66.341, 87.316, -50.83, -113.377]
  MoveL 174 to (34.79, 183.72, 290) mm, rotated rx 180 ry -65 rz 74.51 deg; joints [2.31, 12.298, 1.159, -57.593, 111.853, -85.345, -274.515]
  Set speed (60.0 mm/s)
  MoveL 175 to (31.73, 182.3, 280) mm, rotated rx -180 ry -65 rz 72.21 deg; joints [2.046, 13.71, -1.653, -58.189, 112.379, -86.773, -272.214]
  MoveL 176 to (27.92, 180.74, 270) mm, rotated rx -180 ry -65 rz 69.41 deg; joints [1.78, 14.835, -3.884, -58.69, 112.737, -87.941, -269.407]
  MoveL 177 to (23.38, 179.17, 260) mm, rotated rx -180 ry -65 rz 66.13 deg; joints [1.514, 15.796, -5.783, -59.135, 112.997, -88.96, -266.13]
  MoveL 178 to (18.11, 177.74, 250) mm, rotated rx 180 ry -65 rz 62.42 deg; joints [1.247, 16.646, -7.462, -59.54, 113.193, -89.88, -262.417]
  MoveL 179 to (8.73, 177.85, 238.63) mm, rotated rx -180 ry -65 rz 68.3 deg; joints [0.693, 8.127, 10.028, -57.846, 103.878, -73.23, -258.3]
  MoveL 180 to (5.21, 176.01, 229.84) mm, rotated rx 180 ry -65 rz 63.81 deg; joints [0.427, 8.146, 10.028, -57.958, 103.654, -73.352, -253.813]
  MoveL 181 to (-1.49, 175.64, 220) mm, rotated rx 180 ry -65 rz 58.99 deg; joints [0.16, 11.527, 3.23, -58.818, 105.228, -76.495, -248.987]
  MoveL 182 to (-9.03, 176.15, 210) mm, rotated rx -180 ry -65 rz 53.85 deg; joints [-0.107, 13.112, 0.058, -59.298, 105.821, -78.046, -243.854]
  MoveL 183 to (-16.88, 177.46, 200) mm, rotated rx -180 ry -65 rz 48.44 deg; joints [-0.376, 14.3, -2.314, -59.687, 106.197, -79.246, -238.444]
  MoveL 184 to (-24.89, 179.66, 190) mm, rotated rx -180 ry -65 rz 42.78 deg; joints [-0.645, 15.29, -4.291, -60.03, 106.464, -80.273, -232.785]
  MoveL 185 to (-32.91, 182.83, 180) mm, rotated rx 180 ry -65 rz 36.91 deg; joints [-0.915, 16.155, -6.02, -60.341, 106.663, -81.193, -226.906]
  MoveL 186 to (-40.75, 186.98, 170) mm, rotated rx 180 ry -65 rz 30.84 deg; joints [-1.185, 16.932, -7.574, -60.63, 106.815, -82.037, -220.836]
  MoveL 187 to (-50.04, 195.82, 158.66) mm, rotated rx -180 ry -65 rz 34.6 deg; joints [-1.717, 8.166, 10.028, -60.33, 97.941, -65.614, -214.602]
  MoveL 188 to (-55.54, 199.14, 149.67) mm, rotated rx -180 ry -65 rz 28.23 deg; joints [-1.985, 8.168, 10.028, -60.43, 97.718, -65.739, -208.231]
  MoveL 189 to (-61.48, 205.13, 140) mm, rotated rx -180 ry -65 rz 21.75 deg; joints [-2.255, 11.063, 4.181, -60.903, 98.94, -68.468, -201.752]
  MoveL 190 to (-66.92, 212.81, 130) mm, rotated rx 180 ry -65 rz 15.19 deg; joints [-2.525, 12.722, 0.826, -61.232, 99.531, -70.1, -195.192]
  MoveL 191 to (-71.41, 221.1, 120) mm, rotated rx 180 ry -65 rz 8.58 deg; joints [-2.795, 13.912, -1.584, -61.498, 99.884, -71.314, -188.581]
  MoveL 192 to (-74.87, 229.83, 110) mm, rotated rx 180 ry -65 rz 1.95 deg; joints [-3.067, 14.884, -3.557, -61.731, 100.127, -72.337, -181.949]
  MoveL 193 to (-77.24, 238.83, 100) mm, rotated rx -180 ry -65 rz -4.67 deg; joints [-3.339, 15.723, -5.262, -61.943, 100.3, -73.241, -175.327]
  MoveL 194 to (-78.53, 247.91, 90) mm, rotated rx 180 ry -65 rz -11.25 deg; joints [-3.612, 16.467, -6.778, -62.138, 100.424, -74.061, -168.75]
  MoveL 195 to (-76.26, 262.04, 78.39) mm, rotated rx -180 ry -65 rz -7.75 deg; joints [-4.112, 7.915, 10.028, -63.191, 92.331, -58.03, -162.251]
  MoveL 196 to (-76.48, 268.05, 69.21) mm, rotated rx -180 ry -65 rz -14.13 deg; joints [-4.384, 7.909, 10.028, -63.279, 92.103, -58.152, -155.868]
  MoveL 197 to (-76.32, 274, 59.99) mm, rotated rx 180 ry -65 rz -20.36 deg; joints [-4.656, 7.904, 10.028, -63.367, 91.874, -58.273, -149.641]
  MoveL 198 to (-73.92, 281.75, 50) mm, rotated rx -180 ry -65 rz -26.39 deg; joints [-4.929, 4.626, 16.642, -63.408, 90.149, -55.405, -143.608]
  MoveL 199 to (-70.87, 288.9, 40) mm, rotated rx -180 ry -65 rz -32.19 deg; joints [-5.202, 3.271, 19.373, -63.516, 89.308, -54.288, -137.812]
  MoveL 200 to (-67.34, 295.36, 30) mm, rotated rx -180 ry -65 rz -37.7 deg; joints [-5.477, 2.254, 21.424, -63.639, 88.621, -53.474, -132.296]
  MoveL 201 to (-63.51, 301.08, 20) mm, rotated rx 180 ry -65 rz -42.9 deg; joints [-5.752, 1.414, 23.118, -63.77, 88.017, -52.819, -127.105]
  MoveL 202 to (-59.54, 306.05, 10) mm, rotated rx 180 ry -65 rz -47.72 deg; joints [-6.029, 0.691, 24.58, -63.908, 87.466, -52.265, -122.281]
  MoveL 203 to (-55.59, 310.29, 0) mm, rotated rx -180 ry -65 rz -52.13 deg; joints [-6.306, 0.053, 25.874, -64.052, 86.954, -51.786, -117.87]
  MoveL 204 to (34.79, 183.72, 290) mm, rotated rx 180 ry -65 rz 74.51 deg; joints [2.31, 3.521, 18.897, -54.969, 106.871, -77.447, -274.515]
  Set speed (60.0 mm/s)
  MoveL 205 to (30.72, 204.12, 290) mm, rotated rx -180 ry -65 rz 78.8 deg; joints [2.384, 0.024, 24.728, -54.373, 105.577, -75.423, -278.796]
  MoveL 206 to (-55.59, 310.29, 0) mm, rotated rx -180 ry -65 rz -52.13 deg; joints [-6.306, 0.053, 25.874, -64.052, 86.954, -51.786, -117.87]
  Set speed (60.0 mm/s)
  MoveL 207 to (-44.28, 292.75, -0.25) mm, rotated rx -180 ry -65 rz -35.52 deg; joints [-6.449, 6.917, 10.028, -66.342, 87.305, -50.809, -124.484]
  MoveL 208 to (-55.59, 310.29, 0) mm, rotated rx 180 ry -65 rz -52.13 deg; joints [-6.306, 0.053, 25.874, -64.052, 86.954, -51.786, -117.87]
  Set speed (60.0 mm/s)
  MoveL 209 to (-59.54, 306.05, 10) mm, rotated rx -180 ry -65 rz -47.72 deg; joints [-6.029, 0.691, 24.58, -63.908, 87.466, -52.265, -122.281]
  MoveL 210 to (-63.51, 301.08, 20) mm, rotated rx 180 ry -65 rz -42.9 deg; joints [-5.752, 1.414, 23.118, -63.77, 88.017, -52.819, -127.105]
  MoveL 211 to (-67.34, 295.36, 30) mm, rotated rx -180 ry -65 rz -37.7 deg; joints [-5.477, 2.254, 21.424, -63.639, 88.621, -53.474, -132.296]
  MoveL 212 to (-70.87, 288.9, 40) mm, rotated rx 180 ry -65 rz -32.19 deg; joints [-5.202, 3.271, 19.373, -63.516, 89.308, -54.288, -137.812]
  MoveL 213 to (-73.92, 281.75, 50) mm, rotated rx -180 ry -65 rz -26.39 deg; joints [-4.929, 4.626, 16.642, -63.408, 90.149, -55.405, -143.608]
  MoveL 214 to (-76.32, 274, 59.99) mm, rotated rx -180 ry -65 rz -20.36 deg; joints [-4.656, 7.904, 10.028, -63.367, 91.874, -58.273, -149.641]
  MoveL 215 to (-76.48, 268.05, 69.21) mm, rotated rx 180 ry -65 rz -14.13 deg; joints [-4.384, 7.909, 10.028, -63.279, 92.103, -58.152, -155.868]
  MoveL 216 to (-76.26, 262.04, 78.39) mm, rotated rx -180 ry -65 rz -7.75 deg; joints [-4.112, 7.915, 10.028, -63.191, 92.331, -58.03, -162.251]
  MoveL 217 to (-78.53, 247.91, 90) mm, rotated rx 180 ry -65 rz -11.25 deg; joints [-3.612, -0.164, 26.834, -60.475, 92.225, -59.088, -168.75]
  MoveL 218 to (-77.24, 238.83, 100) mm, rotated rx -180 ry -65 rz -4.67 deg; joints [-3.339, 0.591, 25.318, -60.378, 92.813, -59.629, -175.327]
  MoveL 219 to (-74.87, 229.83, 110) mm, rotated rx 180 ry -65 rz 1.95 deg; joints [-3.067, 1.439, 23.613, -60.295, 93.45, -60.252, -181.949]
  MoveL 220 to (-71.41, 221.1, 120) mm, rotated rx 180 ry -65 rz 8.58 deg; joints [-2.795, 2.42, 21.639, -60.231, 94.157, -60.994, -188.581]
  MoveL 221 to (-66.92, 212.81, 130) mm, rotated rx -180 ry -65 rz 15.19 deg; joints [-2.525, 3.615, 19.23, -60.198, 94.976, -61.928, -195.192]
  MoveL 222 to (-61.48, 205.13, 140) mm, rotated rx -180 ry -65 rz 21.75 deg; joints [-2.255, 5.276, 15.875, -60.227, 96.035, -63.279, -201.752]
  MoveL 223 to (-55.54, 199.14, 149.67) mm, rotated rx -180 ry -65 rz 28.23 deg; joints [-1.985, 8.168, 10.028, -60.43, 97.718, -65.739, -208.231]
  MoveL 224 to (-50.04, 195.82, 158.66) mm, rotated rx 180 ry -65 rz 34.6 deg; joints [-1.717, 8.166, 10.028, -60.33, 97.941, -65.614, -214.602]
  MoveL 225 to (-40.75, 186.98, 170) mm, rotated rx -180 ry -65 rz 30.84 deg; joints [-1.185, 16.932, -7.574, -60.63, 106.815, -82.037, -220.836]
  MoveL 226 to (-32.91, 182.83, 180) mm, rotated rx 180 ry -65 rz 36.91 deg; joints [-0.915, 16.155, -6.02, -60.341, 106.663, -81.193, -226.906]
  MoveL 227 to (-24.89, 179.66, 190) mm, rotated rx 180 ry -65 rz 42.78 deg; joints [-0.645, 15.29, -4.291, -60.03, 106.464, -80.273, -232.785]
  MoveL 228 to (-16.88, 177.46, 200) mm, rotated rx -180 ry -65 rz 48.44 deg; joints [-0.376, 14.3, -2.314, -59.687, 106.197, -79.246, -238.444]
  MoveL 229 to (-9.03, 176.15, 210) mm, rotated rx -180 ry -65 rz 53.85 deg; joints [-0.107, 13.112, 0.058, -59.298, 105.821, -78.046, -243.854]
  MoveL 230 to (-1.49, 175.64, 220) mm, rotated rx -180 ry -65 rz 58.99 deg; joints [0.16, 11.527, 3.23, -58.818, 105.228, -76.495, -248.987]
  MoveL 231 to (5.21, 176.01, 229.84) mm, rotated rx 180 ry -65 rz 63.81 deg; joints [0.427, 8.146, 10.028, -57.958, 103.654, -73.352, -253.813]
  MoveL 232 to (8.73, 177.85, 238.63) mm, rotated rx 180 ry -65 rz 68.3 deg; joints [0.693, 8.127, 10.028, -57.846, 103.878, -73.23, -258.3]
  MoveL 233 to (18.11, 177.74, 250) mm, rotated rx -180 ry -65 rz 62.42 deg; joints [1.247, -0.662, 27.517, -54.579, 103.521, -74.269, -262.417]
  MoveL 234 to (23.38, 179.17, 260) mm, rotated rx -180 ry -65 rz 66.13 deg; joints [1.514, 0.148, 25.839, -54.6, 104.219, -74.855, -266.13]
  MoveL 235 to (27.92, 180.74, 270) mm, rotated rx 180 ry -65 rz 69.41 deg; joints [1.78, 1.067, 23.94, -54.657, 104.983, -75.537, -269.407]
  MoveL 236 to (31.73, 182.3, 280) mm, rotated rx -180 ry -65 rz 72.21 deg; joints [2.046, 2.15, 21.709, -54.768, 105.843, -76.365, -272.214]
  MoveL 237 to (34.79, 183.72, 290) mm, rotated rx 180 ry -65 rz 74.51 deg; joints [2.31, 3.521, 18.897, -54.969, 106.871, -77.447, -274.515]
  MoveL 238 to (30.72, 204.12, 290) mm, rotated rx 180 ry -65 rz 78.8 deg; joints [2.384, 0.024, 24.728, -54.373, 105.577, -75.423, -278.796]
  Set speed (60.0 mm/s)
  MoveL 239 to (28.54, 202.85, 280) mm, rotated rx 180 ry -65 rz 76.53 deg; joints [2.119, -0.875, 26.585, -54.312, 104.823, -74.76, -276.535]
  MoveL 240 to (20.58, 201.82, 267.95) mm, rotated rx -180 ry -65 rz 83.78 deg; joints [1.557, 7.465, 10.028, -57.613, 104.927, -73.354, -273.779]
  MoveL 241 to (20.62, 200.21, 259.26) mm, rotated rx 180 ry -65 rz 80.56 deg; joints [1.293, 7.485, 10.028, -57.723, 104.703, -73.476, -270.563]
  MoveL 242 to (18.7, 198.53, 250) mm, rotated rx 180 ry -65 rz 76.92 deg; joints [1.028, 9.87, 5.249, -58.388, 105.754, -75.721, -266.921]
  MoveL 243 to (14.35, 197.26, 240) mm, rotated rx 180 ry -65 rz 72.89 deg; joints [0.762, 11.875, 1.235, -58.989, 106.578, -77.647, -262.886]
  MoveL 244 to (9.52, 196.26, 230) mm, rotated rx -180 ry -65 rz 68.49 deg; joints [0.495, 13.213, -1.431, -59.431, 107.034, -78.978, -258.492]
  MoveL 245 to (4.24, 195.64, 220) mm, rotated rx -180 ry -65 rz 63.77 deg; joints [0.227, 14.288, -3.569, -59.808, 107.345, -80.077, -253.769]
  MoveL 246 to (-1.41, 195.5, 210) mm, rotated rx 180 ry -65 rz 58.75 deg; joints [-0.041, 15.211, -5.402, -60.146, 107.572, -81.042, -248.748]
  MoveL 247 to (-7.35, 195.94, 200) mm, rotated rx 180 ry -65 rz 53.46 deg; joints [-0.311, 16.032, -7.031, -60.455, 107.742, -81.917, -243.458]
  MoveL 248 to (-17.36, 200.31, 188.25) mm, rotated rx 180 ry -65 rz 57.93 deg; joints [-0.853, 7.552, 10.028, -60.083, 98.959, -65.739, -237.927]
  MoveL 249 to (-21.02, 200.26, 179.33) mm, rotated rx 180 ry -65 rz 52.18 deg; joints [-1.12, 7.562, 10.028, -60.182, 98.733, -65.859, -232.183]
  MoveL 250 to (-25.78, 201.42, 170) mm, rotated rx 180 ry -65 rz 46.25 deg; joints [-1.388, 5.421, 14.371, -60.015, 97.416, -64.059, -226.252]
  MoveL 251 to (-31.7, 204.73, 160) mm, rotated rx 180 ry -65 rz 40.16 deg; joints [-1.657, 3.437, 18.391, -59.915, 96.179, -62.411, -220.159]
  MoveL 252 to (-37.3, 208.79, 150) mm, rotated rx 180 ry -65 rz 33.93 deg; joints [-1.927, 2.139, 21.02, -59.915, 95.296, -61.378, -213.93]
  MoveL 253 to (-42.45, 213.53, 140) mm, rotated rx 180 ry -65 rz 27.59 deg; joints [-2.197, 1.1, 23.123, -59.955, 94.549, -60.579, -207.591]
  MoveL 254 to (-47.02, 218.88, 130) mm, rotated rx 180 ry -65 rz 21.17 deg; joints [-2.468, 0.208, 24.924, -60.019, 93.881, -59.913, -201.168]
  MoveL 255 to (-50.93, 224.75, 120) mm, rotated rx 180 ry -65 rz 14.69 deg; joints [-2.739, -0.584, 26.519, -60.1, 93.268, -59.338, -194.687]
  MoveL 256 to (-54.16, 237.19, 108.16) mm, rotated rx -180 ry -65 rz 18.18 deg; joints [-3.25, 7.351, 10.028, -62.936, 93.319, -58.161, -188.176]
  MoveL 257 to (-56.15, 240.75, 99.06) mm, rotated rx -180 ry -65 rz 11.66 deg; joints [-3.52, 7.346, 10.028, -63.023, 93.092, -58.283, -181.664]
  MoveL 258 to (-58.01, 244.5, 89.93) mm, rotated rx 180 ry -65 rz 5.18 deg; joints [-3.79, 7.339, 10.028, -63.11, 92.865, -58.405, -175.184]
  MoveL 259 to (-58.85, 250.92, 80) mm, rotated rx -180 ry -65 rz -1.23 deg; joints [-4.061, 4.088, 16.585, -63.1, 91.141, -55.572, -168.767]
  MoveL 260 to (-58.87, 257.48, 70) mm, rotated rx -180 ry -65 rz -7.55 deg; joints [-4.333, 2.644, 19.488, -63.184, 90.255, -54.384, -162.451]
  MoveL 261 to (-58.2, 263.79, 60) mm, rotated rx 180 ry -65 rz -13.73 deg; joints [-4.606, 1.566, 21.655, -63.291, 89.541, -53.526, -156.272]
  MoveL 262 to (-56.92, 269.76, 50) mm, rotated rx -180 ry -65 rz -19.73 deg; joints [-4.88, 0.674, 23.444, -63.41, 88.914, -52.836, -150.271]
  MoveL 263 to (-55.13, 275.3, 40) mm, rotated rx -180 ry -65 rz -25.51 deg; joints [-5.154, -0.096, 24.991, -63.538, 88.344, -52.253, -144.491]
  MoveL 264 to (-52.95, 280.35, 30) mm, rotated rx 180 ry -65 rz -31.02 deg; joints [-5.43, -0.778, 26.361, -63.673, 87.814, -51.746, -138.976]
  MoveL 265 to (-45.7, 288.43, 18.51) mm, rotated rx 180 ry -65 rz -26.23 deg; joints [-5.901, 6.92, 10.028, -66.192, 87.784, -50.596, -133.772]
  MoveL 266 to (-44.92, 290.67, 9.15) mm, rotated rx -180 ry -65 rz -31.07 deg; joints [-6.174, 6.917, 10.028, -66.267, 87.545, -50.703, -128.926]
  MoveL 267 to (-44.28, 292.75, -0.25) mm, rotated rx 180 ry -65 rz -35.52 deg; joints [-6.449, 6.917, 10.028, -66.342, 87.305, -50.809, -124.484]
  MoveL 268 to (30.72, 204.12, 290) mm, rotated rx -180 ry -65 rz 78.8 deg; joints [2.384, 14.572, -4.672, -58.835, 113.79, -88.583, -278.796]
  Set speed (60.0 mm/s)
  MoveL 269 to (58.22, 245.2, 290) mm, rotated rx -180 ry -65 rz 125.73 deg; joints [2.398, 14.868, -5.498, -59.031, 114.075, -89.073, -325.735]
  MoveL 270 to (-45.21, 292.27, 0) mm, rotated rx -180 ry -65 rz -55.52 deg; joints [-6.061, 21.696, -18.612, -63.752, 101.26, -81.178, -484.484]
  Set speed (60.0 mm/s)
  MoveL 271 to (-57.47, 247.5, -0.72) mm, rotated rx 180 ry -65 rz 14.89 deg; joints [-6.459, 7.056, 10.028, -66.351, 87.24, -50.686, -534.894]
  MoveL 272 to (-44.28, 292.75, -0.25) mm, rotated rx -180 ry -65 rz -35.52 deg; joints [-6.449, 6.917, 10.028, -66.342, 87.305, -50.809, -484.484]
  Set speed (60.0 mm/s)
  MoveL 273 to (-44.92, 290.67, 9.15) mm, rotated rx 180 ry -65 rz -31.07 deg; joints [-6.174, 6.917, 10.028, -66.267, 87.545, -50.703, -488.926]
  MoveL 274 to (-45.7, 288.43, 18.51) mm, rotated rx -180 ry -65 rz -26.23 deg; joints [-5.901, 6.92, 10.028, -66.192, 87.784, -50.596, -493.772]
  MoveL 275 to (-52.95, 280.35, 30) mm, rotated rx 180 ry -65 rz -31.02 deg; joints [-5.43, -0.778, 26.361, -63.673, 87.814, -51.746, -498.976]
  MoveL 276 to (-55.13, 275.3, 40) mm, rotated rx 180 ry -65 rz -25.51 deg; joints [-5.154, -0.096, 24.991, -63.538, 88.344, -52.253, -504.491]
  MoveL 277 to (-56.92, 269.76, 50) mm, rotated rx 180 ry -65 rz -19.73 deg; joints [-4.88, 0.674, 23.444, -63.41, 88.914, -52.836, -510.271]
  MoveL 278 to (-58.2, 263.79, 60) mm, rotated rx -180 ry -65 rz -13.73 deg; joints [-4.606, 1.566, 21.655, -63.291, 89.541, -53.526, -516.272]
  MoveL 279 to (-58.87, 257.48, 70) mm, rotated rx -180 ry -65 rz -7.55 deg; joints [-4.333, 2.644, 19.488, -63.184, 90.255, -54.384, -522.451]
  MoveL 280 to (-58.85, 250.92, 80) mm, rotated rx -180 ry -65 rz -1.23 deg; joints [-4.061, 4.088, 16.585, -63.1, 91.141, -55.572, -528.767]
  MoveL 281 to (-58.01, 244.5, 89.93) mm, rotated rx 180 ry -65 rz 5.18 deg; joints [-3.79, 7.339, 10.028, -63.11, 92.865, -58.405, -535.184]
  MoveL 282 to (-56.15, 240.75, 99.06) mm, rotated rx -180 ry -65 rz 11.66 deg; joints [-3.52, 7.346, 10.028, -63.023, 93.092, -58.283, -541.664]
  MoveL 283 to (-54.16, 237.19, 108.16) mm, rotated rx -180 ry -65 rz 18.18 deg; joints [-3.25, 7.351, 10.028, -62.936, 93.319, -58.161, -548.176]
  MoveL 284 to (-50.93, 224.75, 120) mm, rotated rx 180 ry -65 rz 14.69 deg; joints [-2.739, -0.584, 26.519, -60.1, 93.268, -59.338, -554.687]
  MoveL 285 to (-47.02, 218.88, 130) mm, rotated rx 180 ry -65 rz 21.17 deg; joints [-2.468, 0.208, 24.924, -60.019, 93.881, -59.913, -561.168]
  MoveL 286 to (-42.45, 213.53, 140) mm, rotated rx 180 ry -65 rz 27.59 deg; joints [-2.197, 1.1, 23.123, -59.955, 94.549, -60.579, -567.591]
  MoveL 287 to (-37.3, 208.79, 150) mm, rotated rx 180 ry -65 rz 33.93 deg; joints [-1.927, 2.139, 21.02, -59.915, 95.296, -61.378, -573.93]
  MoveL 288 to (-31.7, 204.73, 160) mm, rotated rx -180 ry -65 rz 40.16 deg; joints [-1.657, 3.437, 18.391, -59.915, 96.179, -62.411, -580.159]
  MoveL 289 to (-25.78, 201.42, 170) mm, rotated rx -180 ry -65 rz 46.25 deg; joints [-1.388, 5.421, 14.371, -60.015, 97.416, -64.059, -586.252]
  MoveL 290 to (-21.02, 200.26, 179.33) mm, rotated rx 180 ry -65 rz 52.18 deg; joints [-1.12, 7.562, 10.028, -60.182, 98.733, -65.859, -592.183]
  MoveL 291 to (-17.36, 200.31, 188.25) mm, rotated rx 180 ry -65 rz 57.93 deg; joints [-0.853, 7.552, 10.028, -60.083, 98.959, -65.739, -597.927]
  MoveL 292 to (-7.35, 195.94, 200) mm, rotated rx -180 ry -65 rz 53.46 deg; joints [-0.311, -0.851, 27.087, -56.963, 98.736, -66.8, -603.458]
  MoveL 293 to (-1.41, 195.5, 210) mm, rotated rx -180 ry -65 rz 58.75 deg; joints [-0.041, -0.059, 25.458, -56.937, 99.396, -67.377, -608.748]
  MoveL 294 to (4.24, 195.64, 220) mm, rotated rx -180 ry -65 rz 63.77 deg; joints [0.227, 0.832, 23.625, -56.937, 100.114, -68.043, -613.769]
  MoveL 295 to (9.52, 196.26, 230) mm, rotated rx -180 ry -65 rz 68.49 deg; joints [0.495, 1.873, 21.486, -56.974, 100.918, -68.843, -618.492]
  MoveL 296 to (14.35, 197.26, 240) mm, rotated rx -180 ry -65 rz 72.89 deg; joints [0.762, 3.173, 18.82, -57.075, 101.867, -69.875, -622.886]
  MoveL 297 to (18.7, 198.53, 250) mm, rotated rx 180 ry -65 rz 76.92 deg; joints [1.028, 5.14, 14.807, -57.332, 103.185, -71.499, -626.921]
  MoveL 298 to (20.62, 200.21, 259.26) mm, rotated rx 180 ry -65 rz 80.56 deg; joints [1.293, 7.485, 10.028, -57.723, 104.703, -73.476, -630.563]
  MoveL 299 to (20.58, 201.82, 267.95) mm, rotated rx 180 ry -65 rz 83.78 deg; joints [1.557, 7.465, 10.028, -57.613, 104.927, -73.354, -633.779]
  MoveL 300 to (28.54, 202.85, 280) mm, rotated rx -180 ry -65 rz 76.53 deg; joints [2.119, 15.511, -6.529, -59.287, 114.037, -89.592, -636.535]
  MoveL 301 to (30.72, 204.12, 290) mm, rotated rx 180 ry -65 rz 78.8 deg; joints [2.384, 14.572, -4.672, -58.835, 113.79, -88.583, -638.796]
  MoveL 302 to (58.22, 245.2, 290) mm, rotated rx -180 ry -65 rz 125.73 deg; joints [2.398, 14.868, -5.498, -59.031, 114.075, -89.073, -685.735]
  Set speed (60.0 mm/s)
  MoveL 303 to (57.77, 242.72, 280) mm, rotated rx -180 ry -65 rz 123.34 deg; joints [2.132, 15.756, -7.246, -59.464, 114.289, -90.03, -683.345]
  MoveL 304 to (54.25, 237.11, 268.49) mm, rotated rx -180 ry -65 rz 130.44 deg; joints [1.569, 7.362, 10.028, -57.631, 104.992, -73.438, -680.439]
  MoveL 305 to (55.61, 235.88, 259.77) mm, rotated rx -180 ry -65 rz 127.06 deg; joints [1.304, 7.387, 10.028, -57.74, 104.765, -73.556, -677.057]
  MoveL 306 to (54.69, 232.42, 250) mm, rotated rx -180 ry -65 rz 123.24 deg; joints [1.038, 4.153, 16.618, -57.168, 102.747, -70.783, -673.242]
  MoveL 307 to (52.84, 228.29, 240) mm, rotated rx 180 ry -65 rz 119.03 deg; joints [0.771, 2.589, 19.833, -56.996, 101.642, -69.503, -669.031]
  MoveL 308 to (50.46, 223.96, 230) mm, rotated rx 180 ry -65 rz 114.47 deg; joints [0.503, 1.447, 22.197, -56.924, 100.769, -68.596, -664.466]
  MoveL 309 to (47.51, 219.54, 220) mm, rotated rx -180 ry -65 rz 109.58 deg; joints [0.234, 0.509, 24.147, -56.903, 100.01, -67.869, -659.584]
  MoveL 310 to (43.95, 215.15, 210) mm, rotated rx -180 ry -65 rz 104.42 deg; joints [-0.036, -0.3, 25.839, -56.914, 99.324, -67.255, -654.422]
  MoveL 311 to (39.77, 210.92, 200) mm, rotated rx -180 ry -65 rz 99.02 deg; joints [-0.306, -1.021, 27.35, -56.949, 98.689, -66.719, -649.016]
  MoveL 312 to (30.26, 206.52, 188.38) mm, rotated rx -180 ry -65 rz 103.4 deg; joints [-0.85, 7.526, 10.028, -60.085, 98.975, -65.76, -643.399]
  MoveL 313 to (27.77, 203.45, 179.39) mm, rotated rx -180 ry -65 rz 97.6 deg; joints [-1.119, 7.55, 10.028, -60.183, 98.74, -65.869, -637.602]
  MoveL 314 to (23.65, 200.44, 170) mm, rotated rx 180 ry -65 rz 91.66 deg; joints [-1.389, 5.457, 14.302, -60.019, 97.431, -64.087, -631.658]
  MoveL 315 to (17.28, 198.07, 160) mm, rotated rx -180 ry -65 rz 85.59 deg; joints [-1.659, 3.575, 18.146, -59.926, 96.231, -62.504, -625.594]
  MoveL 316 to (10.57, 196.44, 150) mm, rotated rx 180 ry -65 rz 79.44 deg; joints [-1.93, 2.344, 20.673, -59.928, 95.365, -61.504, -619.438]
  MoveL 317 to (3.62, 195.59, 140) mm, rotated rx 180 ry -65 rz 73.22 deg; joints [-2.201, 1.358, 22.698, -59.969, 94.629, -60.726, -613.219]
  MoveL 318 to (-3.42, 195.58, 130) mm, rotated rx -180 ry -65 rz 66.96 deg; joints [-2.474, 0.512, 24.435, -60.033, 93.969, -60.076, -606.961]
  MoveL 319 to (-10.42, 196.41, 120) mm, rotated rx -180 ry -65 rz 60.69 deg; joints [-2.746, -0.24, 25.979, -60.114, 93.36, -59.512, -600.691]
  MoveL 320 to (-17.25, 198.06, 110) mm, rotated rx -180 ry -65 rz 54.44 deg; joints [-3.02, -0.925, 27.381, -60.207, 92.79, -59.011, -594.435]
  MoveL 321 to (-26.77, 204, 98.65) mm, rotated rx 180 ry -65 rz 58.22 deg; joints [-3.529, 7.446, 10.028, -63.021, 93.039, -58.197, -588.22]
  MoveL 322 to (-30.92, 205.13, 89.47) mm, rotated rx 180 ry -65 rz 52.07 deg; joints [-3.8, 7.45, 10.028, -63.109, 92.807, -58.311, -582.072]
  MoveL 323 to (-35.48, 207.36, 80) mm, rotated rx 180 ry -65 rz 46.02 deg; joints [-4.072, 5.506, 13.961, -63.13, 91.677, -56.652, -576.02]
  MoveL 324 to (-40.49, 211.59, 70) mm, rotated rx 180 ry -65 rz 40.09 deg; joints [-4.344, 3.613, 17.788, -63.193, 90.576, -55.042, -570.093]
  MoveL 325 to (-44.86, 216.19, 60) mm, rotated rx 180 ry -65 rz 34.32 deg; joints [-4.617, 2.393, 20.252, -63.293, 89.79, -54.045, -564.321]
  MoveL 326 to (-48.58, 221.03, 50) mm, rotated rx 180 ry -65 rz 28.74 deg; joints [-4.891, 1.424, 22.206, -63.407, 89.123, -53.276, -558.737]
  MoveL 327 to (-51.63, 225.99, 40) mm, rotated rx -180 ry -65 rz 23.38 deg; joints [-5.166, 0.601, 23.867, -63.532, 88.524, -52.64, -553.376]
  MoveL 328 to (-54.06, 230.92, 30) mm, rotated rx -180 ry -65 rz 18.27 deg; joints [-5.441, -0.124, 25.326, -63.665, 87.974, -52.092, -548.272]
  MoveL 329 to (-55.91, 235.73, 20) mm, rotated rx 180 ry -65 rz 13.46 deg; joints [-5.717, -0.773, 26.635, -63.803, 87.459, -51.611, -543.465]
  MoveL 330 to (-56.44, 245.72, 8.66) mm, rotated rx -180 ry -65 rz 18.99 deg; joints [-6.185, 7.058, 10.028, -66.276, 87.479, -50.578, -538.992]
  MoveL 331 to (-57.47, 247.5, -0.72) mm, rotated rx -180 ry -65 rz 14.89 deg; joints [-6.459, 7.056, 10.028, -66.351, 87.24, -50.686, -534.894]
  MoveL 332 to (58.22, 245.2, 290) mm, rotated rx 180 ry -65 rz 125.73 deg; joints [2.398, -0.498, 25.554, -54.297, 105.409, -75.158, -685.735]
  Set speed (60.0 mm/s)
  MoveL 333 to (78.63, 249.2, 290) mm, rotated rx -180 ry -65 rz 132.18 deg; joints [2.326, 2.596, 20.491, -54.795, 106.498, -76.866, -692.181]
  MoveL 334 to (-57.47, 247.5, -0.72) mm, rotated rx 180 ry -65 rz 14.89 deg; joints [-6.459, 7.056, 10.028, -66.351, 87.24, -50.686, -534.894]
  Set speed (60.0 mm/s)
  MoveL 335 to (-76.17, 234.21, 0) mm, rotated rx 180 ry -65 rz 8.7 deg; joints [-6.319, 0.857, 24.584, -64.034, 87.157, -52.228, -538.703]
  MoveL 336 to (-57.47, 247.5, -0.72) mm, rotated rx 180 ry -65 rz 14.89 deg; joints [-6.459, 7.056, 10.028, -66.351, 87.24, -50.686, -534.894]
  Set speed (60.0 mm/s)
  MoveL 337 to (-56.44, 245.72, 8.66) mm, rotated rx 180 ry -65 rz 18.99 deg; joints [-6.185, 7.058, 10.028, -66.276, 87.479, -50.578, -538.992]
  MoveL 338 to (-55.91, 235.73, 20) mm, rotated rx -180 ry -65 rz 13.46 deg; joints [-5.717, -0.773, 26.635, -63.803, 87.459, -51.611, -543.465]
  MoveL 339 to (-54.06, 230.92, 30) mm, rotated rx 180 ry -65 rz 18.27 deg; joints [-5.441, -0.124, 25.326, -63.665, 87.974, -52.092, -548.272]
  MoveL 340 to (-51.63, 225.99, 40) mm, rotated rx -180 ry -65 rz 23.38 deg; joints [-5.166, 0.601, 23.867, -63.532, 88.524, -52.64, -553.376]
  MoveL 341 to (-48.58, 221.03, 50) mm, rotated rx 180 ry -65 rz 28.74 deg; joints [-4.891, 1.424, 22.206, -63.407, 89.123, -53.276, -558.737]
  MoveL 342 to (-44.86, 216.19, 60) mm, rotated rx 180 ry -65 rz 34.32 deg; joints [-4.617, 2.393, 20.252, -63.293, 89.79, -54.045, -564.321]
  MoveL 343 to (-40.49, 211.59, 70) mm, rotated rx 180 ry -65 rz 40.09 deg; joints [-4.344, 3.613, 17.788, -63.193, 90.576, -55.042, -570.093]
  MoveL 344 to (-35.48, 207.36, 80) mm, rotated rx -180 ry -65 rz 46.02 deg; joints [-4.072, 5.506, 13.961, -63.13, 91.677, -56.652, -576.02]
  MoveL 345 to (-30.92, 205.13, 89.47) mm, rotated rx 180 ry -65 rz 52.07 deg; joints [-3.8, 7.45, 10.028, -63.109, 92.807, -58.311, -582.072]
  MoveL 346 to (-26.77, 204, 98.65) mm, rotated rx -180 ry -65 rz 58.22 deg; joints [-3.529, 7.446, 10.028, -63.021, 93.039, -58.197, -588.22]
  MoveL 347 to (-17.25, 198.06, 110) mm, rotated rx 180 ry -65 rz 54.44 deg; joints [-3.02, -0.925, 27.381, -60.207, 92.79, -59.011, -594.435]
  MoveL 348 to (-10.42, 196.41, 120) mm, rotated rx 180 ry -65 rz 60.69 deg; joints [-2.746, -0.24, 25.979, -60.114, 93.36, -59.512, -600.691]
  MoveL 349 to (-3.42, 195.58, 130) mm, rotated rx -180 ry -65 rz 66.96 deg; joints [-2.474, 0.512, 24.435, -60.033, 93.969, -60.076, -606.961]
  MoveL 350 to (3.62, 195.59, 140) mm, rotated rx -180 ry -65 rz 73.22 deg; joints [-2.201, 1.358, 22.698, -59.969, 94.629, -60.726, -613.219]
  MoveL 351 to (10.57, 196.44, 150) mm, rotated rx 180 ry -65 rz 79.44 deg; joints [-1.93, 2.344, 20.673, -59.928, 95.365, -61.504, -619.438]
  MoveL 352 to (17.28, 198.07, 160) mm, rotated rx -180 ry -65 rz 85.59 deg; joints [-1.659, 3.575, 18.146, -59.926, 96.231, -62.504, -625.594]
  MoveL 353 to (23.65, 200.44, 170) mm, rotated rx 180 ry -65 rz 91.66 deg; joints [-1.389, 5.457, 14.302, -60.019, 97.431, -64.087, -631.658]
  MoveL 354 to (27.77, 203.45, 179.39) mm, rotated rx -180 ry -65 rz 97.6 deg; joints [-1.119, 7.55, 10.028, -60.183, 98.74, -65.869, -637.602]
  MoveL 355 to (30.26, 206.52, 188.38) mm, rotated rx -180 ry -65 rz 103.4 deg; joints [-0.85, 7.526, 10.028, -60.085, 98.975, -65.76, -643.399]
  MoveL 356 to (39.77, 210.92, 200) mm, rotated rx -180 ry -65 rz 99.02 deg; joints [-0.306, 16.122, -7.295, -60.502, 107.831, -82.073, -649.016]
  MoveL 357 to (43.95, 215.15, 210) mm, rotated rx -180 ry -65 rz 104.42 deg; joints [-0.036, 15.347, -5.783, -60.211, 107.698, -81.262, -654.422]
  MoveL 358 to (47.51, 219.54, 220) mm, rotated rx 180 ry -65 rz 109.58 deg; joints [0.234, 14.483, -4.091, -59.895, 107.516, -80.371, -659.584]
  MoveL 359 to (50.46, 223.96, 230) mm, rotated rx -180 ry -65 rz 114.47 deg; joints [0.503, 13.491, -2.141, -59.544, 107.261, -79.365, -664.466]
  MoveL 360 to (52.84, 228.29, 240) mm, rotated rx 180 ry -65 rz 119.03 deg; joints [0.771, 12.293, 0.223, -59.139, 106.892, -78.175, -669.031]
  MoveL 361 to (54.69, 232.42, 250) mm, rotated rx 180 ry -65 rz 123.24 deg; joints [1.038, 10.675, 3.438, -58.63, 106.289, -76.608, -673.242]
  MoveL 362 to (55.61, 235.88, 259.77) mm, rotated rx -180 ry -65 rz 127.06 deg; joints [1.304, 7.387, 10.028, -57.74, 104.765, -73.556, -677.057]
  MoveL 363 to (54.25, 237.11, 268.49) mm, rotated rx -180 ry -65 rz 130.44 deg; joints [1.569, 7.362, 10.028, -57.631, 104.992, -73.438, -680.439]
  MoveL 364 to (57.77, 242.72, 280) mm, rotated rx -180 ry -65 rz 123.34 deg; joints [2.132, 15.756, -7.246, -59.464, 114.289, -90.03, -683.345]
  MoveL 365 to (58.22, 245.2, 290) mm, rotated rx -180 ry -65 rz 125.73 deg; joints [2.398, 14.868, -5.498, -59.031, 114.075, -89.073, -685.735]
  MoveL 366 to (78.63, 249.2, 290) mm, rotated rx -180 ry -65 rz 132.18 deg; joints [2.326, 12.952, -0.436, -57.909, 112.369, -86.195, -692.181]
  Set speed (60.0 mm/s)
  MoveL 367 to (78.34, 245.85, 280) mm, rotated rx -180 ry -65 rz 129.76 deg; joints [2.061, 14.182, -2.871, -58.447, 112.785, -87.452, -689.758]
  MoveL 368 to (77.78, 241.77, 270) mm, rotated rx -180 ry -65 rz 126.81 deg; joints [1.795, 15.203, -4.882, -58.912, 113.076, -88.518, -686.809]
  MoveL 369 to (76.86, 237.05, 260) mm, rotated rx 180 ry -65 rz 123.37 deg; joints [1.528, 16.092, -6.624, -59.329, 113.288, -89.461, -683.374]
  MoveL 370 to (71.4, 228.23, 247.95) mm, rotated rx 180 ry -65 rz 129.49 deg; joints [0.971, 7.998, 10.028, -57.752, 104.17, -73.197, -679.493]
  MoveL 371 to (71.69, 224.69, 239.15) mm, rotated rx 180 ry -65 rz 125.21 deg; joints [0.704, 8.027, 10.028, -57.862, 103.941, -73.311, -675.208]
  MoveL 372 to (70.88, 219.99, 230) mm, rotated rx -180 ry -65 rz 120.56 deg; joints [0.437, 9.876, 6.351, -58.372, 104.689, -75.052, -670.555]
  MoveL 373 to (67.49, 213.75, 220) mm, rotated rx -180 ry -65 rz 115.58 deg; joints [0.169, 12.05, 2.017, -58.978, 105.591, -77.103, -665.575]
  MoveL 374 to (63.28, 207.47, 210) mm, rotated rx 180 ry -65 rz 110.31 deg; joints [-0.101, 13.403, -0.658, -59.4, 106.043, -78.423, -660.305]
  MoveL 375 to (58.22, 201.33, 200) mm, rotated rx -180 ry -65 rz 104.78 deg; joints [-0.371, 14.473, -2.762, -59.755, 106.34, -79.491, -654.781]
  MoveL 376 to (52.31, 195.49, 190) mm, rotated rx 180 ry -65 rz 99.04 deg; joints [-0.641, 15.386, -4.55, -60.07, 106.548, -80.418, -649.037]
  MoveL 377 to (45.56, 190.13, 180) mm, rotated rx -180 ry -65 rz 93.11 deg; joints [-0.913, 16.193, -6.127, -60.359, 106.699, -81.254, -643.107]
  MoveL 378 to (38.04, 185.42, 170) mm, rotated rx 180 ry -65 rz 87.02 deg; joints [-1.185, 16.924, -7.553, -60.626, 106.808, -82.024, -637.024]
  MoveL 379 to (25.47, 182.1, 158.56) mm, rotated rx -180 ry -65 rz 90.82 deg; joints [-1.719, 8.187, 10.028, -60.328, 97.929, -65.596, -630.818]
  MoveL 380 to (19.57, 178.89, 149.49) mm, rotated rx 180 ry -65 rz 84.52 deg; joints [-1.989, 8.208, 10.028, -60.427, 97.695, -65.706, -624.519]
  MoveL 381 to (11.96, 176.54, 140) mm, rotated rx -180 ry -65 rz 78.16 deg; joints [-2.26, 5.982, 14.565, -60.286, 96.33, -63.81, -618.157]
  MoveL 382 to (2.59, 175.67, 130) mm, rotated rx -180 ry -65 rz 71.76 deg; joints [-2.532, 4.195, 18.208, -60.235, 95.189, -62.315, -611.758]
  MoveL 383 to (-6.83, 175.92, 120) mm, rotated rx -180 ry -65 rz 65.35 deg; joints [-2.804, 2.994, 20.663, -60.261, 94.349, -61.347, -605.352]
  MoveL 384 to (-16.13, 177.3, 110) mm, rotated rx -180 ry -65 rz 58.97 deg; joints [-3.077, 2.026, 22.644, -60.32, 93.632, -60.59, -598.967]
  MoveL 385 to (-25.11, 179.73, 100) mm, rotated rx -180 ry -65 rz 52.63 deg; joints [-3.35, 1.193, 24.347, -60.399, 92.986, -59.955, -592.629]
  MoveL 386 to (-33.62, 183.16, 90) mm, rotated rx 180 ry -65 rz 46.37 deg; joints [-3.624, 0.451, 25.861, -60.493, 92.391, -59.404, -586.369]
  MoveL 387 to (-41.52, 187.45, 80) mm, rotated rx -180 ry -65 rz 40.21 deg; joints [-3.899, -0.224, 27.235, -60.599, 91.834, -58.915, -580.214]
  MoveL 388 to (-50.92, 197.05, 68.6) mm, rotated rx 180 ry -65 rz 44.2 deg; joints [-4.397, 8.061, 10.028, -63.279, 92.024, -58.022, -574.197]
  MoveL 389 to (-55.89, 200.31, 59.36) mm, rotated rx -180 ry -65 rz 38.35 deg; joints [-4.669, 8.062, 10.028, -63.367, 91.792, -58.137, -568.347]
  MoveL 390 to (-60.61, 204.07, 50) mm, rotated rx -180 ry -65 rz 32.7 deg; joints [-4.942, 9.171, 7.788, -63.487, 92.065, -59.266, -562.698]
  MoveL 391 to (-65.29, 210.3, 40) mm, rotated rx -180 ry -65 rz 27.28 deg; joints [-5.216, 11.485, 3.111, -63.658, 92.881, -61.501, -557.284]
  MoveL 392 to (-69.12, 216.58, 30) mm, rotated rx 180 ry -65 rz 22.14 deg; joints [-5.491, 12.756, 0.54, -63.793, 93.217, -62.786, -552.14]
  MoveL 393 to (-72.16, 222.75, 20) mm, rotated rx -180 ry -65 rz 17.3 deg; joints [-5.766, 13.734, -1.438, -63.913, 93.417, -63.804, -547.303]
  MoveL 394 to (-74.48, 228.68, 10) mm, rotated rx -180 ry -65 rz 12.81 deg; joints [-6.042, 14.552, -3.091, -64.022, 93.541, -64.675, -542.811]
  MoveL 395 to (-76.17, 234.21, 0) mm, rotated rx -180 ry -65 rz 8.7 deg; joints [-6.319, 15.262, -4.528, -64.124, 93.614, -65.448, -538.703]
  MoveL 396 to (78.63, 249.2, 290) mm, rotated rx 180 ry -65 rz 132.18 deg; joints [2.326, 12.952, -0.436, -57.909, 112.369, -86.195, -692.181]
  Set speed (60.0 mm/s)
  MoveL 397 to (58.93, 255.88, 290) mm, rotated rx 180 ry -65 rz 136 deg; joints [2.402, 14.944, -5.714, -59.083, 114.15, -89.202, -695.998]
  MoveL 398 to (-76.17, 234.21, 0) mm, rotated rx 180 ry -65 rz 8.7 deg; joints [-6.319, 15.262, -4.528, -64.124, 93.614, -65.448, -538.703]
  Set speed (60.0 mm/s)
  MoveL 399 to (-55.23, 237.63, -0.82) mm, rotated rx -180 ry -65 rz 24.99 deg; joints [-6.461, 7.085, 10.028, -66.353, 87.227, -50.66, -544.986]
  MoveL 400 to (-76.17, 234.21, 0) mm, rotated rx 180 ry -65 rz 8.7 deg; joints [-6.319, 0.857, 24.584, -64.034, 87.157, -52.228, -538.703]
  Set speed (60.0 mm/s)
  MoveL 401 to (-74.48, 228.68, 10) mm, rotated rx -180 ry -65 rz 12.81 deg; joints [-6.042, 1.568, 23.147, -63.893, 87.701, -52.771, -542.811]
  MoveL 402 to (-72.16, 222.75, 20) mm, rotated rx -180 ry -65 rz 17.3 deg; joints [-5.766, 2.386, 21.494, -63.757, 88.295, -53.409, -547.303]
  MoveL 403 to (-69.12, 216.58, 30) mm, rotated rx -180 ry -65 rz 22.14 deg; joints [-5.491, 3.366, 19.516, -63.629, 88.963, -54.192, -552.14]
  MoveL 404 to (-65.29, 210.3, 40) mm, rotated rx 180 ry -65 rz 27.28 deg; joints [-5.216, 4.639, 16.945, -63.513, 89.769, -55.242, -557.284]
  MoveL 405 to (-60.61, 204.07, 50) mm, rotated rx 180 ry -65 rz 32.7 deg; joints [-4.942, 6.954, 12.268, -63.432, 91.053, -57.241, -562.698]
  MoveL 406 to (-55.89, 200.31, 59.36) mm, rotated rx 180 ry -65 rz 38.35 deg; joints [-4.669, 8.062, 10.028, -63.367, 91.792, -58.137, -568.347]
  MoveL 407 to (-50.92, 197.05, 68.6) mm, rotated rx -180 ry -65 rz 44.2 deg; joints [-4.397, 8.061, 10.028, -63.279, 92.024, -58.022, -574.197]
  MoveL 408 to (-41.52, 187.45, 80) mm, rotated rx 180 ry -65 rz 40.21 deg; joints [-3.899, 16.805, -7.179, -62.221, 100.204, -74.252, -580.214]
  MoveL 409 to (-33.62, 183.16, 90) mm, rotated rx 180 ry -65 rz 46.37 deg; joints [-3.624, 16.12, -5.805, -62.041, 100.121, -73.505, -586.369]
  MoveL 410 to (-25.11, 179.73, 100) mm, rotated rx 180 ry -65 rz 52.63 deg; joints [-3.35, 15.364, -4.291, -61.849, 100.002, -72.697, -592.629]
  MoveL 411 to (-16.13, 177.3, 110) mm, rotated rx 180 ry -65 rz 58.97 deg; joints [-3.077, 14.512, -2.588, -61.641, 99.835, -71.807, -598.967]
  MoveL 412 to (-6.83, 175.92, 120) mm, rotated rx 180 ry -65 rz 65.35 deg; joints [-2.804, 13.52, -0.607, -61.412, 99.597, -70.797, -605.352]
  MoveL 413 to (2.59, 175.67, 130) mm, rotated rx -180 ry -65 rz 71.76 deg; joints [-2.532, 12.291, 1.848, -61.149, 99.24, -69.578, -611.758]
  MoveL 414 to (11.96, 176.54, 140) mm, rotated rx 180 ry -65 rz 78.16 deg; joints [-2.26, 10.472, 5.491, -60.808, 98.585, -67.835, -618.157]
  MoveL 415 to (19.57, 178.89, 149.49) mm, rotated rx 180 ry -65 rz 84.52 deg; joints [-1.989, 8.208, 10.028, -60.427, 97.695, -65.706, -624.519]
  MoveL 416 to (25.47, 182.1, 158.56) mm, rotated rx 180 ry -65 rz 90.82 deg; joints [-1.719, 8.187, 10.028, -60.328, 97.929, -65.596, -630.818]
  MoveL 417 to (38.04, 185.42, 170) mm, rotated rx 180 ry -65 rz 87.02 deg; joints [-1.185, -0.475, 27.609, -57.308, 97.592, -66.466, -637.024]
  MoveL 418 to (45.56, 190.13, 180) mm, rotated rx -180 ry -65 rz 93.11 deg; joints [-0.913, 0.205, 26.183, -57.255, 98.2, -66.967, -643.107]
  MoveL 419 to (52.31, 195.49, 190) mm, rotated rx -180 ry -65 rz 99.04 deg; joints [-0.641, 0.959, 24.605, -57.22, 98.852, -67.534, -649.037]
  MoveL 420 to (58.22, 201.33, 200) mm, rotated rx 180 ry -65 rz 104.78 deg; joints [-0.371, 1.815, 22.818, -57.21, 99.562, -68.193, -654.781]
  MoveL 421 to (63.28, 207.47, 210) mm, rotated rx -180 ry -65 rz 110.31 deg; joints [-0.101, 2.827, 20.713, -57.238, 100.36, -68.99, -660.305]
  MoveL 422 to (67.49, 213.75, 220) mm, rotated rx -180 ry -65 rz 115.58 deg; joints [0.169, 4.121, 18.039, -57.33, 101.315, -70.036, -665.575]
  MoveL 423 to (70.88, 219.99, 230) mm, rotated rx 180 ry -65 rz 120.56 deg; joints [0.437, 6.237, 13.705, -57.603, 102.72, -71.811, -670.555]
  MoveL 424 to (71.69, 224.69, 239.15) mm, rotated rx -180 ry -65 rz 125.21 deg; joints [0.704, 8.027, 10.028, -57.862, 103.941, -73.311, -675.208]
  MoveL 425 to (71.4, 228.23, 247.95) mm, rotated rx 180 ry -65 rz 129.49 deg; joints [0.971, 7.998, 10.028, -57.752, 104.17, -73.197, -679.493]
  MoveL 426 to (76.86, 237.05, 260) mm, rotated rx -180 ry -65 rz 123.37 deg; joints [1.528, -0.388, 26.68, -54.529, 104.052, -74.591, -683.374]
  MoveL 427 to (77.78, 241.77, 270) mm, rotated rx -180 ry -65 rz 126.81 deg; joints [1.795, 0.447, 24.938, -54.567, 104.775, -75.21, -686.809]
  MoveL 428 to (78.34, 245.85, 280) mm, rotated rx -180 ry -65 rz 129.76 deg; joints [2.061, 1.416, 22.927, -54.648, 105.575, -75.946, -689.758]
  MoveL 429 to (78.63, 249.2, 290) mm, rotated rx -180 ry -65 rz 132.18 deg; joints [2.326, 2.596, 20.491, -54.795, 106.498, -76.866, -692.181]
  MoveL 430 to (58.93, 255.88, 290) mm, rotated rx -180 ry -65 rz 136 deg; joints [2.402, -0.635, 25.77, -54.277, 105.366, -75.09, -695.998]
  Set speed (60.0 mm/s)
  MoveL 431 to (58.94, 253.36, 280) mm, rotated rx 180 ry -65 rz 133.57 deg; joints [2.136, -1.465, 27.495, -54.235, 104.649, -74.483, -693.568]
  MoveL 432 to (56.71, 247.53, 268.65) mm, rotated rx 180 ry -65 rz 140.62 deg; joints [1.573, 7.332, 10.028, -57.636, 105.011, -73.462, -690.615]
  MoveL 433 to (58.3, 246.54, 259.92) mm, rotated rx -180 ry -65 rz 137.18 deg; joints [1.307, 7.358, 10.028, -57.745, 104.783, -73.579, -687.181]
  MoveL 434 to (57.77, 242.68, 250) mm, rotated rx 180 ry -65 rz 133.31 deg; joints [1.041, 3.892, 17.088, -57.127, 102.637, -70.601, -683.306]
  MoveL 435 to (56.69, 238.28, 240) mm, rotated rx 180 ry -65 rz 129.03 deg; joints [0.774, 2.407, 20.146, -56.972, 101.573, -69.39, -679.034]
  MoveL 436 to (55.14, 233.59, 230) mm, rotated rx 180 ry -65 rz 124.41 deg; joints [0.506, 1.3, 22.441, -56.907, 100.718, -68.512, -674.405]
  MoveL 437 to (53.04, 228.71, 220) mm, rotated rx -180 ry -65 rz 119.46 deg; joints [0.237, 0.386, 24.347, -56.891, 99.971, -67.804, -669.46]
  MoveL 438 to (50.33, 223.75, 210) mm, rotated rx 180 ry -65 rz 114.24 deg; joints [-0.033, -0.406, 26.006, -56.905, 99.293, -67.202, -664.235]
  MoveL 439 to (46.98, 218.83, 200) mm, rotated rx -180 ry -65 rz 108.77 deg; joints [-0.304, -1.112, 27.49, -56.941, 98.664, -66.676, -658.769]
  MoveL 440 to (38.67, 212.91, 188.47) mm, rotated rx -180 ry -65 rz 113.1 deg; joints [-0.848, 7.507, 10.028, -60.087, 98.986, -65.776, -653.096]
  MoveL 441 to (36.76, 209.37, 179.47) mm, rotated rx -180 ry -65 rz 107.25 deg; joints [-1.117, 7.534, 10.028, -60.185, 98.75, -65.882, -647.251]
  MoveL 442 to (33.03, 205.6, 170) mm, rotated rx 180 ry -65 rz 101.26 deg; joints [-1.387, 9.848, 5.402, -60.607, 99.667, -68.048, -641.263]
  MoveL 443 to (27.19, 202.13, 160) mm, rotated rx -180 ry -65 rz 95.16 deg; joints [-1.658, 11.673, 1.76, -60.976, 100.324, -69.788, -635.164]
  MoveL 444 to (20.88, 199.3, 150) mm, rotated rx -180 ry -65 rz 88.98 deg; joints [-1.929, 12.911, -0.698, -61.258, 100.682, -71.004, -628.983]
  MoveL 445 to (14.2, 197.22, 140) mm, rotated rx -180 ry -65 rz 82.75 deg; joints [-2.201, 13.912, -2.681, -61.502, 100.919, -72.012, -622.746]
  MoveL 446 to (7.28, 195.93, 130) mm, rotated rx 180 ry -65 rz 76.48 deg; joints [-2.474, 14.773, -4.387, -61.723, 101.085, -72.898, -616.481]
  MoveL 447 to (0.24, 195.48, 120) mm, rotated rx -180 ry -65 rz 70.21 deg; joints [-2.747, 15.54, -5.906, -61.926, 101.203, -73.704, -610.213]
  MoveL 448 to (-6.77, 195.87, 110) mm, rotated rx 180 ry -65 rz 63.97 deg; joints [-3.02, 16.235, -7.287, -62.116, 101.286, -74.45, -603.969]
  MoveL 449 to (-17.27, 200.13, 98.61) mm, rotated rx -180 ry -65 rz 67.78 deg; joints [-3.529, 7.454, 10.028, -63.021, 93.034, -58.19, -597.775]
  MoveL 450 to (-21.59, 200.49, 89.43) mm, rotated rx 180 ry -65 rz 61.66 deg; joints [-3.801, 7.462, 10.028, -63.108, 92.8, -58.301, -591.658]
  MoveL 451 to (-26.38, 201.72, 80) mm, rotated rx -180 ry -65 rz 55.64 deg; joints [-4.073, 9.183, 6.56, -63.276, 93.355, -59.98, -585.644]
  MoveL 452 to (-32.08, 204.97, 70) mm, rotated rx -180 ry -65 rz 49.76 deg; joints [-4.346, 11.178, 2.535, -63.47, 94.029, -61.916, -579.763]
  MoveL 453 to (-37.21, 208.71, 60) mm, rotated rx 180 ry -65 rz 44.04 deg; joints [-4.619, 12.418, 0.034, -63.624, 94.353, -63.168, -574.043]
  MoveL 454 to (-41.73, 212.8, 50) mm, rotated rx -180 ry -65 rz 38.52 deg; joints [-4.893, 13.394, -1.938, -63.759, 94.554, -64.182, -568.517]
  MoveL 455 to (-45.64, 217.12, 40) mm, rotated rx -180 ry -65 rz 33.22 deg; joints [-5.168, 14.22, -3.608, -63.883, 94.684, -65.061, -563.217]
  MoveL 456 to (-48.92, 221.54, 30) mm, rotated rx 180 ry -65 rz 28.18 deg; joints [-5.443, 14.945, -5.074, -63.996, 94.766, -65.849, -558.176]
  MoveL 457 to (-51.6, 225.93, 20) mm, rotated rx -180 ry -65 rz 23.43 deg; joints [-5.719, 15.595, -6.389, -64.102, 94.812, -66.569, -553.433]
  MoveL 458 to (-53.91, 236.06, 8.57) mm, rotated rx 180 ry -65 rz 29.02 deg; joints [-6.187, 7.086, 10.028, -66.277, 87.466, -50.554, -549.023]
  MoveL 459 to (-55.23, 237.63, -0.82) mm, rotated rx 180 ry -65 rz 24.99 deg; joints [-6.461, 7.085, 10.028, -66.353, 87.227, -50.66, -544.986]
  MoveL 460 to (58.93, 255.88, 290) mm, rotated rx -180 ry -65 rz 136 deg; joints [2.402, 14.944, -5.714, -59.083, 114.15, -89.202, -695.998]
  Set speed (60.0 mm/s)
  MoveL 461 to (37.11, 300.24, 290) mm, rotated rx -180 ry -65 rz -172.69 deg; joints [2.418, 15.257, -6.615, -59.305, 114.465, -89.748, -747.315]
  MoveL 462 to (-55.37, 234.2, 0) mm, rotated rx -180 ry -65 rz 4.99 deg; joints [-6.074, 21.523, -17.912, -63.66, 101.015, -80.702, -904.986]
  Set speed (60.0 mm/s)
  MoveL 463 to (-23.82, 202.61, -1.14) mm, rotated rx -180 ry -65 rz 71.39 deg; joints [-6.468, 7.179, 10.028, -66.359, 87.183, -50.576, -951.385]
  MoveL 464 to (-55.23, 237.63, -0.82) mm, rotated rx 180 ry -65 rz 24.99 deg; joints [-6.461, 7.085, 10.028, -66.353, 87.227, -50.66, -904.986]
  Set speed (60.0 mm/s)
  MoveL 465 to (-53.91, 236.06, 8.57) mm, rotated rx 180 ry -65 rz 29.02 deg; joints [-6.187, 7.086, 10.028, -66.277, 87.466, -50.554, -909.023]
  MoveL 466 to (-51.6, 225.93, 20) mm, rotated rx -180 ry -65 rz 23.43 deg; joints [-5.719, 15.595, -6.389, -64.102, 94.812, -66.569, -913.433]
  MoveL 467 to (-48.92, 221.54, 30) mm, rotated rx -180 ry -65 rz 28.18 deg; joints [-5.443, 14.945, -5.074, -63.996, 94.766, -65.849, -918.176]
  MoveL 468 to (-45.64, 217.12, 40) mm, rotated rx -180 ry -65 rz 33.22 deg; joints [-5.168, 14.22, -3.608, -63.883, 94.684, -65.061, -923.217]
  MoveL 469 to (-41.73, 212.8, 50) mm, rotated rx 180 ry -65 rz 38.52 deg; joints [-4.893, 13.394, -1.938, -63.759, 94.554, -64.182, -928.517]
  MoveL 470 to (-37.21, 208.71, 60) mm, rotated rx -180 ry -65 rz 44.04 deg; joints [-4.619, 12.418, 0.034, -63.624, 94.353, -63.168, -934.043]
  MoveL 471 to (-32.08, 204.97, 70) mm, rotated rx -180 ry -65 rz 49.76 deg; joints [-4.346, 11.178, 2.535, -63.47, 94.029, -61.916, -939.763]
  MoveL 472 to (-26.38, 201.72, 80) mm, rotated rx 180 ry -65 rz 55.64 deg; joints [-4.073, 9.183, 6.56, -63.276, 93.355, -59.98, -945.644]
  MoveL 473 to (-21.59, 200.49, 89.43) mm, rotated rx 180 ry -65 rz 61.66 deg; joints [-3.801, 7.462, 10.028, -63.108, 92.8, -58.301, -951.658]
  MoveL 474 to (-17.27, 200.13, 98.61) mm, rotated rx -180 ry -65 rz 67.78 deg; joints [-3.529, 7.454, 10.028, -63.021, 93.034, -58.19, -957.775]
  MoveL 475 to (-6.77, 195.87, 110) mm, rotated rx -180 ry -65 rz 63.97 deg; joints [-3.02, -0.9, 27.343, -60.208, 92.797, -59.023, -963.969]
  MoveL 476 to (0.24, 195.48, 120) mm, rotated rx 180 ry -65 rz 70.21 deg; joints [-2.747, -0.229, 25.961, -60.114, 93.363, -59.517, -970.213]
  MoveL 477 to (7.28, 195.93, 130) mm, rotated rx -180 ry -65 rz 76.48 deg; joints [-2.474, 0.507, 24.442, -60.033, 93.967, -60.073, -976.481]
  MoveL 478 to (14.2, 197.22, 140) mm, rotated rx 180 ry -65 rz 82.75 deg; joints [-2.201, 1.334, 22.736, -59.968, 94.622, -60.712, -982.746]
  MoveL 479 to (20.88, 199.3, 150) mm, rotated rx 180 ry -65 rz 88.98 deg; joints [-1.929, 2.296, 20.754, -59.925, 95.349, -61.474, -988.983]
  MoveL 480 to (27.19, 202.13, 160) mm, rotated rx 180 ry -65 rz 95.16 deg; joints [-1.658, 3.491, 18.296, -59.92, 96.199, -62.447, -995.164]
  MoveL 481 to (33.03, 205.6, 170) mm, rotated rx -180 ry -65 rz 101.26 deg; joints [-1.387, 5.269, 14.654, -60, 97.351, -63.943, -1001.263]
  MoveL 482 to (36.76, 209.37, 179.47) mm, rotated rx 180 ry -65 rz 107.25 deg; joints [-1.117, 7.534, 10.028, -60.185, 98.75, -65.882, -1007.251]
  MoveL 483 to (38.67, 212.91, 188.47) mm, rotated rx -180 ry -65 rz 113.1 deg; joints [-0.848, 7.507, 10.028, -60.087, 98.986, -65.776, -1013.096]
  MoveL 484 to (46.98, 218.83, 200) mm, rotated rx 180 ry -65 rz 108.77 deg; joints [-0.304, 16.17, -7.434, -60.527, 107.878, -82.156, -1018.769]
  MoveL 485 to (50.33, 223.75, 210) mm, rotated rx -180 ry -65 rz 114.24 deg; joints [-0.033, 15.406, -5.95, -60.24, 107.754, -81.359, -1024.235]
  MoveL 486 to (53.04, 228.71, 220) mm, rotated rx -180 ry -65 rz 119.46 deg; joints [0.237, 14.557, -4.291, -59.928, 107.581, -80.484, -1029.46]
  MoveL 487 to (55.14, 233.59, 230) mm, rotated rx -180 ry -65 rz 124.41 deg; joints [0.506, 13.584, -2.385, -59.583, 107.339, -79.498, -1034.405]
  MoveL 488 to (56.69, 238.28, 240) mm, rotated rx 180 ry -65 rz 129.03 deg; joints [0.774, 12.42, -0.09, -59.186, 106.989, -78.34, -1039.034]
  MoveL 489 to (57.77, 242.68, 250) mm, rotated rx -180 ry -65 rz 133.31 deg; joints [1.041, 10.879, 2.968, -58.695, 106.43, -76.843, -1043.306]
  MoveL 490 to (58.3, 246.54, 259.92) mm, rotated rx 180 ry -65 rz 137.18 deg; joints [1.307, 7.358, 10.028, -57.745, 104.783, -73.579, -1047.181]
  MoveL 491 to (56.71, 247.53, 268.65) mm, rotated rx 180 ry -65 rz 140.62 deg; joints [1.573, 7.332, 10.028, -57.636, 105.011, -73.462, -1050.615]
  MoveL 492 to (58.94, 253.36, 280) mm, rotated rx 180 ry -65 rz 133.57 deg; joints [2.136, 15.821, -7.439, -59.513, 114.357, -90.149, -1053.568]
  MoveL 493 to (58.93, 255.88, 290) mm, rotated rx -180 ry -65 rz 136 deg; joints [2.402, 14.944, -5.714, -59.083, 114.15, -89.202, -1055.998]
  MoveL 494 to (37.11, 300.24, 290) mm, rotated rx -180 ry -65 rz -172.69 deg; joints [2.418, 15.257, -6.615, -59.305, 114.465, -89.748, -1107.315]
  Set speed (60.0 mm/s)
  MoveL 495 to (40.48, 293.86, 278.03) mm, rotated rx -180 ry -65 rz -165.31 deg; joints [1.852, 7.174, 10.028, -57.55, 105.321, -73.452, -1104.686]
  MoveL 496 to (41.68, 294.92, 269.36) mm, rotated rx -180 ry -65 rz -168.51 deg; joints [1.589, 7.196, 10.028, -57.66, 105.097, -73.573, -1101.487]
  MoveL 497 to (43.78, 293.91, 260) mm, rotated rx -180 ry -65 rz -172.23 deg; joints [1.324, 4.628, 15.266, -57.206, 103.448, -71.391, -1097.765]
  MoveL 498 to (46.4, 290.79, 250) mm, rotated rx 180 ry -65 rz -176.43 deg; joints [1.057, 2.782, 19.046, -56.962, 102.188, -69.864, -1093.565]
  MoveL 499 to (49.06, 287.12, 240) mm, rotated rx 180 ry -65 rz 178.94 deg; joints [0.79, 1.539, 21.612, -56.862, 101.259, -68.869, -1088.935]
  MoveL 500 to (51.62, 282.9, 230) mm, rotated rx -180 ry -65 rz 173.92 deg; joints [0.522, 0.549, 23.669, -56.825, 100.469, -68.097, -1083.922]
  MoveL 501 to (53.98, 278.14, 220) mm, rotated rx -180 ry -65 rz 168.57 deg; joints [0.253, -0.288, 25.421, -56.824, 99.764, -67.455, -1078.571]
  MoveL 502 to (56, 272.86, 210) mm, rotated rx 180 ry -65 rz 162.93 deg; joints [-0.018, -1.021, 26.964, -56.85, 99.116, -66.903, -1072.931]
  MoveL 503 to (55.62, 261.97, 198.07) mm, rotated rx -180 ry -65 rz 167.05 deg; joints [-0.565, 7.345, 10.028, -60.003, 99.3, -65.782, -1067.046]
  MoveL 504 to (57.38, 258.61, 189.08) mm, rotated rx -180 ry -65 rz 160.96 deg; joints [-0.835, 7.377, 10.028, -60.1, 99.062, -65.884, -1060.96]
  MoveL 505 to (58.95, 254.55, 180) mm, rotated rx -180 ry -65 rz 154.71 deg; joints [-1.105, 8.169, 8.495, -60.303, 99.206, -66.665, -1054.714]
  MoveL 506 to (58.59, 247.92, 170) mm, rotated rx -180 ry -65 rz 148.35 deg; joints [-1.375, 10.866, 3.11, -60.799, 100.3, -69.17, -1048.348]
  MoveL 507 to (57.45, 241.22, 160) mm, rotated rx 180 ry -65 rz 141.9 deg; joints [-1.647, 12.24, 0.401, -61.102, 100.717, -70.488, -1041.898]
  MoveL 508 to (55.51, 234.59, 150) mm, rotated rx -180 ry -65 rz 135.4 deg; joints [-1.92, 13.298, -1.673, -61.354, 100.973, -71.525, -1035.4]
  MoveL 509 to (52.77, 228.15, 140) mm, rotated rx -180 ry -65 rz 128.88 deg; joints [-2.193, 14.19, -3.411, -61.578, 101.141, -72.413, -1028.885]
  MoveL 510 to (49.26, 222.05, 130) mm, rotated rx -180 ry -65 rz 122.38 deg; joints [-2.467, 14.974, -4.934, -61.781, 101.255, -73.206, -1022.384]
  MoveL 511 to (45.04, 216.4, 120) mm, rotated rx -180 ry -65 rz 115.93 deg; joints [-2.741, 15.681, -6.304, -61.97, 101.329, -73.933, -1015.926]
  MoveL 512 to (40.19, 211.31, 110) mm, rotated rx 180 ry -65 rz 109.54 deg; joints [-3.016, 16.329, -7.558, -62.146, 101.373, -74.609, -1009.537]
  MoveL 513 to (30.47, 206.45, 98.72) mm, rotated rx 180 ry -65 rz 113.24 deg; joints [-3.527, 7.429, 10.028, -63.022, 93.048, -58.212, -1003.245]
  MoveL 514 to (27.22, 203.17, 89.47) mm, rotated rx 180 ry -65 rz 107.07 deg; joints [-3.8, 7.451, 10.028, -63.109, 92.806, -58.31, -997.074]
  MoveL 515 to (23.03, 200.17, 80) mm, rotated rx 180 ry -65 rz 101.05 deg; joints [-4.073, 5.824, 13.357, -63.138, 91.805, -56.908, -991.051]
  MoveL 516 to (16.86, 197.94, 70) mm, rotated rx -180 ry -65 rz 95.2 deg; joints [-4.347, 3.925, 17.229, -63.197, 90.685, -55.263, -985.201]
  MoveL 517 to (10.69, 196.46, 60) mm, rotated rx -180 ry -65 rz 89.55 deg; joints [-4.622, 2.748, 19.64, -63.294, 89.902, -54.276, -979.549]
  MoveL 518 to (4.64, 195.67, 50) mm, rotated rx -180 ry -65 rz 84.12 deg; joints [-4.897, 1.819, 21.545, -63.406, 89.237, -53.517, -974.124]
  MoveL 519 to (-1.18, 195.49, 40) mm, rotated rx -180 ry -65 rz 78.95 deg; joints [-5.172, 1.03, 23.165, -63.529, 88.641, -52.887, -968.952]
  MoveL 520 to (-6.67, 195.86, 30) mm, rotated rx -180 ry -65 rz 74.06 deg; joints [-5.449, 0.334, 24.593, -63.659, 88.09, -52.343, -964.062]
  MoveL 521 to (-11.76, 196.67, 20) mm, rotated rx 180 ry -65 rz 69.48 deg; joints [-5.725, -0.294, 25.879, -63.796, 87.574, -51.862, -959.483]
  MoveL 522 to (-16.38, 197.8, 10) mm, rotated rx -180 ry -65 rz 65.25 deg; joints [-6.003, -0.867, 27.054, -63.937, 87.085, -51.432, -955.247]
  MoveL 523 to (-23.82, 202.61, -1.14) mm, rotated rx 180 ry -65 rz 71.39 deg; joints [-6.468, 7.179, 10.028, -66.359, 87.183, -50.576, -951.385]
  MoveL 524 to (37.11, 300.24, 290) mm, rotated rx -180 ry -65 rz -172.69 deg; joints [2.418, -1.215, 26.671, -54.196, 105.19, -74.811, -1107.315]
  Set speed (60.0 mm/s)
  MoveL 525 to (43.85, 319.91, 290) mm, rotated rx -180 ry -65 rz -166.2 deg; joints [2.345, 1.666, 22.057, -54.633, 106.146, -76.315, -1113.803]
  MoveL 526 to (-23.82, 202.61, -1.14) mm, rotated rx -180 ry -65 rz 71.39 deg; joints [-6.468, 7.179, 10.028, -66.359, 87.183, -50.576, -951.385]
  Set speed (60.0 mm/s)
  MoveL 527 to (-20.57, 178.36, 0) mm, rotated rx 180 ry -65 rz 65.86 deg; joints [-6.327, 14.897, -3.558, -64.093, 93.342, -64.907, -955.856]
  MoveL 528 to (-23.82, 202.61, -1.14) mm, rotated rx 180 ry -65 rz 71.39 deg; joints [-6.468, 7.179, 10.028, -66.359, 87.183, -50.576, -951.385]
  Set speed (60.0 mm/s)
  MoveL 529 to (-16.38, 197.8, 10) mm, rotated rx 180 ry -65 rz 65.25 deg; joints [-6.003, 15.983, -6.998, -64.174, 94.657, -66.891, -955.247]
  MoveL 530 to (-11.76, 196.67, 20) mm, rotated rx -180 ry -65 rz 69.48 deg; joints [-5.725, 15.394, -5.823, -64.076, 94.648, -66.242, -959.483]
  MoveL 531 to (-6.67, 195.86, 30) mm, rotated rx -180 ry -65 rz 74.06 deg; joints [-5.449, 14.748, -4.537, -63.973, 94.612, -65.545, -964.062]
  MoveL 532 to (-1.18, 195.49, 40) mm, rotated rx 180 ry -65 rz 78.95 deg; joints [-5.172, 14.031, -3.109, -63.861, 94.543, -64.784, -968.952]
  MoveL 533 to (4.64, 195.67, 50) mm, rotated rx 180 ry -65 rz 84.12 deg; joints [-4.897, 13.218, -1.489, -63.741, 94.43, -63.939, -974.124]
  MoveL 534 to (10.69, 196.46, 60) mm, rotated rx -180 ry -65 rz 89.55 deg; joints [-4.622, 12.261, 0.416, -63.609, 94.25, -62.967, -979.549]
  MoveL 535 to (16.86, 197.94, 70) mm, rotated rx 180 ry -65 rz 95.2 deg; joints [-4.347, 11.053, 2.827, -63.46, 93.954, -61.768, -985.201]
  MoveL 536 to (23.03, 200.17, 80) mm, rotated rx -180 ry -65 rz 101.05 deg; joints [-4.073, 9.118, 6.699, -63.273, 93.322, -59.913, -991.051]
  MoveL 537 to (27.22, 203.17, 89.47) mm, rotated rx 180 ry -65 rz 107.07 deg; joints [-3.8, 7.451, 10.028, -63.109, 92.806, -58.31, -997.074]
  MoveL 538 to (30.47, 206.45, 98.72) mm, rotated rx -180 ry -65 rz 113.24 deg; joints [-3.527, 7.429, 10.028, -63.022, 93.048, -58.212, -1003.245]
  MoveL 539 to (40.19, 211.31, 110) mm, rotated rx 180 ry -65 rz 109.54 deg; joints [-3.016, -1.076, 27.614, -60.202, 92.752, -58.938, -1009.537]
  MoveL 540 to (45.04, 216.4, 120) mm, rotated rx 180 ry -65 rz 115.93 deg; joints [-2.741, -0.482, 26.36, -60.104, 93.295, -59.389, -1015.926]
  MoveL 541 to (49.26, 222.05, 130) mm, rotated rx -180 ry -65 rz 122.38 deg; joints [-2.467, 0.167, 24.99, -60.017, 93.87, -59.891, -1022.384]
  MoveL 542 to (52.77, 228.15, 140) mm, rotated rx 180 ry -65 rz 128.88 deg; joints [-2.193, 0.89, 23.467, -59.944, 94.485, -60.46, -1028.885]
  MoveL 543 to (55.51, 234.59, 150) mm, rotated rx -180 ry -65 rz 135.4 deg; joints [-1.92, 1.718, 21.729, -59.889, 95.157, -61.125, -1035.4]
  MoveL 544 to (57.45, 241.22, 160) mm, rotated rx -180 ry -65 rz 141.9 deg; joints [-1.647, 2.712, 19.655, -59.862, 95.916, -61.937, -1041.898]
  MoveL 545 to (58.59, 247.92, 170) mm, rotated rx 180 ry -65 rz 148.35 deg; joints [-1.375, 4.02, 16.946, -59.883, 96.838, -63.029, -1048.348]
  MoveL 546 to (58.95, 254.55, 180) mm, rotated rx 180 ry -65 rz 154.71 deg; joints [-1.105, 6.651, 11.561, -60.094, 98.437, -65.305, -1054.714]
  MoveL 547 to (57.38, 258.61, 189.08) mm, rotated rx -180 ry -65 rz 160.96 deg; joints [-0.835, 7.377, 10.028, -60.1, 99.062, -65.884, -1060.96]
  MoveL 548 to (55.62, 261.97, 198.07) mm, rotated rx 180 ry -65 rz 167.05 deg; joints [-0.565, 7.345, 10.028, -60.003, 99.3, -65.782, -1067.046]
  MoveL 549 to (56, 272.86, 210) mm, rotated rx -180 ry -65 rz 162.93 deg; joints [-0.018, 15.741, -6.909, -60.411, 108.076, -81.921, -1072.931]
  MoveL 550 to (53.98, 278.14, 220) mm, rotated rx -180 ry -65 rz 168.57 deg; joints [0.253, 14.946, -5.365, -60.113, 107.937, -81.098, -1078.571]
  MoveL 551 to (51.62, 282.9, 230) mm, rotated rx -180 ry -65 rz 173.92 deg; joints [0.522, 14.05, -3.613, -59.785, 107.738, -80.181, -1083.922]
  MoveL 552 to (49.06, 287.12, 240) mm, rotated rx -180 ry -65 rz 178.94 deg; joints [0.79, 13.004, -1.557, -59.416, 107.454, -79.126, -1088.935]
  MoveL 553 to (46.4, 290.79, 250) mm, rotated rx -180 ry -65 rz -176.43 deg; joints [1.057, 11.707, 1.01, -58.98, 107.028, -77.844, -1093.565]
  MoveL 554 to (43.78, 293.91, 260) mm, rotated rx -180 ry -65 rz -172.23 deg; joints [1.324, 9.812, 4.79, -58.395, 106.269, -76.023, -1097.765]
  MoveL 555 to (41.68, 294.92, 269.36) mm, rotated rx -180 ry -65 rz -168.51 deg; joints [1.589, 7.196, 10.028, -57.66, 105.097, -73.573, -1101.487]
  MoveL 556 to (40.48, 293.86, 278.03) mm, rotated rx -180 ry -65 rz -165.31 deg; joints [1.852, 7.174, 10.028, -57.55, 105.321, -73.452, -1104.686]
  MoveL 557 to (37.11, 300.24, 290) mm, rotated rx -180 ry -65 rz -172.69 deg; joints [2.418, -1.215, 26.671, -54.196, 105.19, -74.811, -1107.315]
  MoveL 558 to (43.85, 319.91, 290) mm, rotated rx -180 ry -65 rz -166.2 deg; joints [2.345, 1.666, 22.057, -54.633, 106.146, -76.315, -1113.803]
  Set speed (60.0 mm/s)
  MoveL 559 to (46.6, 317.98, 280) mm, rotated rx -180 ry -65 rz -168.79 deg; joints [2.081, 0.601, 24.252, -54.522, 105.294, -75.504, -1111.207]
  MoveL 560 to (49.86, 315.46, 270) mm, rotated rx -180 ry -65 rz -171.95 deg; joints [1.815, -0.301, 26.122, -54.463, 104.536, -74.833, -1108.046]
  MoveL 561 to (53.49, 312.31, 260) mm, rotated rx -180 ry -65 rz -175.64 deg; joints [1.547, -1.092, 27.769, -54.44, 103.843, -74.258, -1104.36]
  MoveL 562 to (58, 305.42, 248.82) mm, rotated rx -180 ry -65 rz -169.81 deg; joints [0.99, 7.833, 10.028, -57.779, 104.274, -73.331, -1100.194]
  MoveL 563 to (61.34, 303.9, 240) mm, rotated rx -180 ry -65 rz -174.41 deg; joints [0.723, 8.292, 9.155, -57.984, 104.279, -73.833, -1095.591]
  MoveL 564 to (65.27, 298.59, 230) mm, rotated rx -180 ry -65 rz -179.4 deg; joints [0.456, 11.471, 2.787, -58.821, 105.731, -76.784, -1090.596]
  MoveL 565 to (68.98, 292.54, 220) mm, rotated rx -180 ry -65 rz 175.25 deg; joints [0.187, 12.942, -0.125, -59.277, 106.248, -78.209, -1085.253]
  MoveL 566 to (72.31, 285.76, 210) mm, rotated rx -180 ry -65 rz 169.61 deg; joints [-0.082, 14.064, -2.33, -59.648, 106.572, -79.321, -1079.605]
  MoveL 567 to (75.1, 278.3, 200) mm, rotated rx 180 ry -65 rz 163.7 deg; joints [-0.353, 15.004, -4.163, -59.972, 106.791, -80.267, -1073.697]
  MoveL 568 to (77.2, 270.26, 190) mm, rotated rx 180 ry -65 rz 157.57 deg; joints [-0.625, 15.825, -5.755, -60.265, 106.944, -81.104, -1067.571]
  MoveL 569 to (78.47, 261.74, 180) mm, rotated rx -180 ry -65 rz 151.27 deg; joints [-0.897, 16.561, -7.174, -60.533, 107.047, -81.863, -1061.269]
  MoveL 570 to (75.86, 248.47, 168.24) mm, rotated rx -180 ry -65 rz 154.83 deg; joints [-1.435, 8.025, 10.028, -60.24, 98.243, -65.603, -1054.829]
  MoveL 571 to (76.41, 241.84, 159.15) mm, rotated rx -180 ry -65 rz 148.29 deg; joints [-1.706, 8.06, 10.028, -60.338, 98.002, -65.702, -1048.29]
  MoveL 572 to (76.31, 234.75, 150) mm, rotated rx 180 ry -65 rz 141.69 deg; joints [-1.978, 8.618, 8.968, -60.501, 98.025, -66.271, -1041.689]
  MoveL 573 to (73.44, 225.85, 140) mm, rotated rx -180 ry -65 rz 135.06 deg; joints [-2.251, 11.418, 3.377, -60.964, 99.161, -68.863, -1035.058]
  MoveL 574 to (69.5, 217.29, 130) mm, rotated rx -180 ry -65 rz 128.43 deg; joints [-2.524, 12.771, 0.708, -61.242, 99.565, -70.16, -1028.432]
  MoveL 575 to (64.57, 209.26, 120) mm, rotated rx -180 ry -65 rz 121.84 deg; joints [-2.798, 13.812, -1.333, -61.475, 99.81, -71.18, -1021.84]
  MoveL 576 to (58.74, 201.9, 110) mm, rotated rx -180 ry -65 rz 115.31 deg; joints [-3.072, 14.689, -3.046, -61.683, 99.972, -72.056, -1015.313]
  MoveL 577 to (52.14, 195.34, 100) mm, rotated rx -180 ry -65 rz 108.88 deg; joints [-3.347, 15.46, -4.549, -61.874, 100.081, -72.841, -1008.879]
  MoveL 578 to (44.91, 189.68, 90) mm, rotated rx -180 ry -65 rz 102.57 deg; joints [-3.623, 16.156, -5.904, -62.051, 100.151, -73.561, -1002.567]
  MoveL 579 to (37.24, 184.98, 80) mm, rotated rx -180 ry -65 rz 96.4 deg; joints [-3.899, 16.793, -7.145, -62.217, 100.193, -74.232, -996.403]
  MoveL 580 to (23.94, 182.03, 68.51) mm, rotated rx -180 ry -65 rz 100.42 deg; joints [-4.399, 8.083, 10.028, -63.279, 92.012, -58.003, -990.416]
  MoveL 581 to (18.4, 179.25, 59.2) mm, rotated rx -180 ry -65 rz 94.63 deg; joints [-4.673, 8.101, 10.028, -63.367, 91.771, -58.104, -984.633]
  MoveL 582 to (12.84, 176.92, 49.87) mm, rotated rx 180 ry -65 rz 89.08 deg; joints [-4.947, 8.117, 10.028, -63.455, 91.531, -58.206, -979.083]
  MoveL 583 to (5.58, 175.83, 40) mm, rotated rx 180 ry -65 rz 83.79 deg; joints [-5.222, 5.364, 15.621, -63.514, 90.031, -55.78, -973.794]
  MoveL 584 to (-1.77, 175.65, 30) mm, rotated rx 180 ry -65 rz 78.8 deg; joints [-5.497, 3.995, 18.411, -63.624, 89.169, -54.621, -968.796]
  MoveL 585 to (-8.64, 176.1, 20) mm, rotated rx 180 ry -65 rz 74.12 deg; joints [-5.773, 2.992, 20.462, -63.749, 88.477, -53.795, -964.119]
  MoveL 586 to (-14.93, 177.06, 10) mm, rotated rx -180 ry -65 rz 69.79 deg; joints [-6.05, 2.165, 22.152, -63.882, 87.869, -53.131, -959.795]
  MoveL 587 to (-20.57, 178.36, 0) mm, rotated rx -180 ry -65 rz 65.86 deg; joints [-6.327, 1.451, 23.614, -64.022, 87.314, -52.57, -955.856]
  MoveL 588 to (43.85, 319.91, 290) mm, rotated rx -180 ry -65 rz -166.2 deg; joints [2.345, 1.666, 22.057, -54.633, 106.146, -76.315, -1113.803]
  Set speed (60.0 mm/s)
  MoveL 589 to (28.22, 306.19, 290) mm, rotated rx -180 ry -65 rz -161.42 deg; joints [2.42, -1.294, 26.794, -54.186, 105.166, -74.773, -1118.582]
  MoveL 590 to (-20.57, 178.36, 0) mm, rotated rx 180 ry -65 rz 65.86 deg; joints [-6.327, 1.451, 23.614, -64.022, 87.314, -52.57, -955.856]
  Set speed (60.0 mm/s)
  MoveL 591 to (-14.1, 199.28, -1.17) mm, rotated rx -180 ry -65 rz 80.93 deg; joints [-6.469, 7.186, 10.028, -66.36, 87.179, -50.57, -960.929]
  MoveL 592 to (-20.57, 178.36, 0) mm, rotated rx -180 ry -65 rz 65.86 deg; joints [-6.327, 14.897, -3.558, -64.093, 93.342, -64.907, -955.856]
  Set speed (60.0 mm/s)
  MoveL 593 to (-14.93, 177.06, 10) mm, rotated rx -180 ry -65 rz 69.79 deg; joints [-6.05, 14.165, -2.096, -63.992, 93.267, -64.131, -959.795]
  MoveL 594 to (-8.64, 176.1, 20) mm, rotated rx -180 ry -65 rz 74.12 deg; joints [-5.773, 13.319, -0.406, -63.883, 93.139, -63.253, -964.119]
  MoveL 595 to (-1.77, 175.65, 30) mm, rotated rx 180 ry -65 rz 78.8 deg; joints [-5.497, 12.293, 1.645, -63.764, 92.928, -62.213, -968.796]
  MoveL 596 to (5.58, 175.83, 40) mm, rotated rx 180 ry -65 rz 83.79 deg; joints [-5.222, 10.899, 4.435, -63.628, 92.548, -60.841, -973.794]
  MoveL 597 to (12.84, 176.92, 49.87) mm, rotated rx 180 ry -65 rz 89.08 deg; joints [-4.947, 8.117, 10.028, -63.455, 91.531, -58.206, -979.083]
  MoveL 598 to (18.4, 179.25, 59.2) mm, rotated rx 180 ry -65 rz 94.63 deg; joints [-4.673, 8.101, 10.028, -63.367, 91.771, -58.104, -984.633]
  MoveL 599 to (23.94, 182.03, 68.51) mm, rotated rx -180 ry -65 rz 100.42 deg; joints [-4.399, 8.083, 10.028, -63.279, 92.012, -58.003, -990.416]
  MoveL 600 to (37.24, 184.98, 80) mm, rotated rx -180 ry -65 rz 96.4 deg; joints [-3.899, -0.202, 27.201, -60.599, 91.839, -58.926, -996.403]
  MoveL 601 to (44.91, 189.68, 90) mm, rotated rx 180 ry -65 rz 102.57 deg; joints [-3.623, 0.389, 25.96, -60.491, 92.374, -59.372, -1002.567]
  MoveL 602 to (52.14, 195.34, 100) mm, rotated rx -180 ry -65 rz 108.88 deg; joints [-3.347, 1.034, 24.605, -60.394, 92.94, -59.867, -1008.879]
  MoveL 603 to (58.74, 201.9, 110) mm, rotated rx -180 ry -65 rz 115.31 deg; joints [-3.072, 1.75, 23.102, -60.308, 93.545, -60.429, -1015.313]
  MoveL 604 to (64.57, 209.26, 120) mm, rotated rx -180 ry -65 rz 121.84 deg; joints [-2.798, 2.568, 21.389, -60.239, 94.206, -61.084, -1021.84]
  MoveL 605 to (69.5, 217.29, 130) mm, rotated rx -180 ry -65 rz 128.43 deg; joints [-2.524, 3.547, 19.348, -60.194, 94.952, -61.883, -1028.432]
  MoveL 606 to (73.44, 225.85, 140) mm, rotated rx 180 ry -65 rz 135.06 deg; joints [-2.251, 4.835, 16.679, -60.192, 95.858, -62.96, -1035.058]
  MoveL 607 to (76.31, 234.75, 150) mm, rotated rx -180 ry -65 rz 141.69 deg; joints [-1.978, 7.569, 11.088, -60.374, 97.497, -65.331, -1041.689]
  MoveL 608 to (76.41, 241.84, 159.15) mm, rotated rx 180 ry -65 rz 148.29 deg; joints [-1.706, 8.06, 10.028, -60.338, 98.002, -65.702, -1048.29]
  MoveL 609 to (75.86, 248.47, 168.24) mm, rotated rx -180 ry -65 rz 154.83 deg; joints [-1.435, 8.025, 10.028, -60.24, 98.243, -65.603, -1054.829]
  MoveL 610 to (78.47, 261.74, 180) mm, rotated rx 180 ry -65 rz 151.27 deg; joints [-0.897, 16.561, -7.174, -60.533, 107.047, -81.863, -1061.269]
  MoveL 611 to (77.2, 270.26, 190) mm, rotated rx -180 ry -65 rz 157.57 deg; joints [-0.625, 15.825, -5.755, -60.265, 106.944, -81.104, -1067.571]
  MoveL 612 to (75.1, 278.3, 200) mm, rotated rx -180 ry -65 rz 163.7 deg; joints [-0.353, 15.004, -4.163, -59.972, 106.791, -80.267, -1073.697]
  MoveL 613 to (72.31, 285.76, 210) mm, rotated rx -180 ry -65 rz 169.61 deg; joints [-0.082, 14.064, -2.33, -59.648, 106.572, -79.321, -1079.605]
  MoveL 614 to (68.98, 292.54, 220) mm, rotated rx 180 ry -65 rz 175.25 deg; joints [0.187, 12.942, -0.125, -59.277, 106.248, -78.209, -1085.253]
  MoveL 615 to (65.27, 298.59, 230) mm, rotated rx -180 ry -65 rz -179.4 deg; joints [0.456, 11.471, 2.787, -58.821, 105.731, -76.784, -1090.596]
  MoveL 616 to (61.34, 303.9, 240) mm, rotated rx 180 ry -65 rz -174.41 deg; joints [0.723, 8.292, 9.155, -57.984, 104.279, -73.833, -1095.591]
  MoveL 617 to (58, 305.42, 248.82) mm, rotated rx 180 ry -65 rz -169.81 deg; joints [0.99, 7.833, 10.028, -57.779, 104.274, -73.331, -1100.194]
  MoveL 618 to (53.49, 312.31, 260) mm, rotated rx -180 ry -65 rz -175.64 deg; joints [1.547, -1.092, 27.769, -54.44, 103.843, -74.258, -1104.36]
  MoveL 619 to (49.86, 315.46, 270) mm, rotated rx -180 ry -65 rz -171.95 deg; joints [1.815, -0.301, 26.122, -54.463, 104.536, -74.833, -1108.046]
  MoveL 620 to (46.6, 317.98, 280) mm, rotated rx -180 ry -65 rz -168.79 deg; joints [2.081, 0.601, 24.252, -54.522, 105.294, -75.504, -1111.207]
  MoveL 621 to (43.85, 319.91, 290) mm, rotated rx -180 ry -65 rz -166.2 deg; joints [2.345, 1.666, 22.057, -54.633, 106.146, -76.315, -1113.803]
  MoveL 622 to (28.22, 306.19, 290) mm, rotated rx -180 ry -65 rz -161.42 deg; joints [2.42, -1.294, 26.794, -54.186, 105.166, -74.773, -1118.582]
  Set speed (60.0 mm/s)
  MoveL 623 to (32.63, 300.8, 278.13) mm, rotated rx -180 ry -65 rz -154.08 deg; joints [1.855, 7.155, 10.028, -57.554, 105.334, -73.468, -1115.919]
  MoveL 624 to (33.57, 302.05, 269.47) mm, rotated rx -180 ry -65 rz -157.32 deg; joints [1.591, 7.175, 10.028, -57.664, 105.11, -73.59, -1112.679]
  MoveL 625 to (35.92, 301.18, 260) mm, rotated rx -180 ry -65 rz -161.09 deg; joints [1.326, 10.015, 4.334, -58.457, 106.404, -76.246, -1108.905]
  MoveL 626 to (39.07, 298.58, 250) mm, rotated rx -180 ry -65 rz -165.36 deg; joints [1.06, 11.827, 0.719, -59.024, 107.118, -77.996, -1104.643]
  MoveL 627 to (42.34, 295.45, 240) mm, rotated rx -180 ry -65 rz -170.06 deg; joints [0.793, 13.099, -1.799, -59.455, 107.531, -79.258, -1099.941]
  MoveL 628 to (45.62, 291.76, 230) mm, rotated rx 180 ry -65 rz -175.15 deg; joints [0.525, 14.131, -3.832, -59.822, 107.81, -80.304, -1094.846]
  MoveL 629 to (48.8, 287.5, 220) mm, rotated rx -180 ry -65 rz 179.41 deg; joints [0.256, 15.019, -5.57, -60.149, 108.005, -81.217, -1089.406]
  MoveL 630 to (51.74, 282.68, 210) mm, rotated rx 180 ry -65 rz 173.67 deg; joints [-0.015, 15.807, -7.102, -60.446, 108.142, -82.036, -1083.668]
  MoveL 631 to (53.44, 272.3, 198.22) mm, rotated rx 180 ry -65 rz 177.68 deg; joints [-0.562, 7.315, 10.028, -60.006, 99.318, -65.806, -1077.679]
  MoveL 632 to (55.81, 269.32, 189.23) mm, rotated rx -180 ry -65 rz 171.49 deg; joints [-0.831, 7.347, 10.028, -60.103, 99.08, -65.909, -1071.486]
  MoveL 633 to (57.96, 265.2, 180) mm, rotated rx -180 ry -65 rz 165.13 deg; joints [-1.101, 5.868, 13.081, -60.001, 98.071, -64.658, -1065.13]
  MoveL 634 to (58.8, 258.62, 170) mm, rotated rx 180 ry -65 rz 158.66 deg; joints [-1.372, 3.749, 17.431, -59.859, 96.733, -62.841, -1058.655]
  MoveL 635 to (58.89, 251.83, 160) mm, rotated rx -180 ry -65 rz 152.1 deg; joints [-1.644, 2.509, 20.004, -59.847, 95.845, -61.808, -1052.098]
  MoveL 636 to (58.18, 244.95, 150) mm, rotated rx 180 ry -65 rz 145.5 deg; joints [-1.917, 1.551, 22.008, -59.879, 95.103, -61.026, -1045.497]
  MoveL 637 to (56.65, 238.12, 140) mm, rotated rx -180 ry -65 rz 138.89 deg; joints [-2.19, 0.746, 23.7, -59.937, 94.442, -60.381, -1038.886]
  MoveL 638 to (54.3, 231.49, 130) mm, rotated rx 180 ry -65 rz 132.3 deg; joints [-2.464, 0.043, 25.187, -60.012, 93.835, -59.826, -1032.295]
  MoveL 639 to (51.17, 225.17, 120) mm, rotated rx 180 ry -65 rz 125.76 deg; joints [-2.739, -0.589, 26.527, -60.1, 93.267, -59.335, -1025.756]
  MoveL 640 to (47.33, 219.29, 110) mm, rotated rx 180 ry -65 rz 119.3 deg; joints [-3.014, -1.167, 27.755, -60.199, 92.729, -58.894, -1019.296]
  MoveL 641 to (38.89, 212.87, 98.8) mm, rotated rx 180 ry -65 rz 122.94 deg; joints [-3.525, 7.41, 10.028, -63.022, 93.058, -58.228, -1012.941]
  MoveL 642 to (36.26, 208.99, 89.54) mm, rotated rx -180 ry -65 rz 116.72 deg; joints [-3.798, 7.435, 10.028, -63.109, 92.814, -58.324, -1006.718]
  MoveL 643 to (32.46, 205.23, 80) mm, rotated rx 180 ry -65 rz 110.65 deg; joints [-4.072, 9.32, 6.264, -63.284, 93.427, -60.121, -1000.653]
  MoveL 644 to (26.8, 201.92, 70) mm, rotated rx 180 ry -65 rz 104.77 deg; joints [-4.346, 11.124, 2.66, -63.466, 93.997, -61.853, -994.769]
  MoveL 645 to (21, 199.35, 60) mm, rotated rx 180 ry -65 rz 99.09 deg; joints [-4.621, 12.299, 0.325, -63.613, 94.275, -63.014, -989.094]
  MoveL 646 to (15.19, 197.47, 50) mm, rotated rx 180 ry -65 rz 93.65 deg; joints [-4.896, 13.237, -1.537, -63.743, 94.443, -63.965, -983.653]
  MoveL 647 to (9.5, 196.25, 40) mm, rotated rx -180 ry -65 rz 88.47 deg; joints [-5.172, 14.038, -3.127, -63.862, 94.548, -64.794, -978.473]
  MoveL 648 to (4.03, 195.62, 30) mm, rotated rx 180 ry -65 rz 83.58 deg; joints [-5.449, 14.747, -4.532, -63.972, 94.611, -65.542, -973.581]
  MoveL 649 to (-1.12, 195.49, 20) mm, rotated rx -180 ry -65 rz 79.01 deg; joints [-5.726, 15.386, -5.801, -64.075, 94.641, -66.229, -969.007]
  MoveL 650 to (-5.87, 195.78, 10) mm, rotated rx 180 ry -65 rz 74.78 deg; joints [-6.003, 15.97, -6.961, -64.172, 94.646, -66.869, -964.779]
  MoveL 651 to (-14.1, 199.28, -1.17) mm, rotated rx 180 ry -65 rz 80.93 deg; joints [-6.469, 7.186, 10.028, -66.36, 87.179, -50.57, -960.929]
  MoveL 652 to (28.22, 306.19, 290) mm, rotated rx 180 ry -65 rz -161.42 deg; joints [2.42, 15.299, -6.738, -59.336, 114.508, -89.823, -1118.582]
  Set speed (60.0 mm/s)
  MoveL 653 to (-21.11, 309.47, 290) mm, rotated rx -180 ry -65 rz -106.89 deg; joints [2.421, 15.322, -6.805, -59.353, 114.532, -89.864, -1173.11]
  MoveL 654 to (-10.16, 196.36, 0) mm, rotated rx 180 ry -65 rz 70.93 deg; joints [-6.281, 16.51, -8.033, -64.263, 94.63, -67.47, -1320.929]
  Set speed (60.0 mm/s)
  MoveL 655 to (33.26, 208.35, -1.05) mm, rotated rx 180 ry -65 rz 126.44 deg; joints [-6.466, 7.153, 10.028, -66.357, 87.195, -50.6, -1366.442]
  MoveL 656 to (-14.1, 199.28, -1.17) mm, rotated rx 180 ry -65 rz 80.93 deg; joints [-6.469, 7.186, 10.028, -66.36, 87.179, -50.57, -1320.929]
  Set speed (60.0 mm/s)
  MoveL 657 to (-5.87, 195.78, 10) mm, rotated rx -180 ry -65 rz 74.78 deg; joints [-6.003, 15.97, -6.961, -64.172, 94.646, -66.869, -1324.779]
  MoveL 658 to (-1.12, 195.49, 20) mm, rotated rx 180 ry -65 rz 79.01 deg; joints [-5.726, 15.386, -5.801, -64.075, 94.641, -66.229, -1329.007]
  MoveL 659 to (4.03, 195.62, 30) mm, rotated rx 180 ry -65 rz 83.58 deg; joints [-5.449, 14.747, -4.532, -63.972, 94.611, -65.542, -1333.581]
  MoveL 660 to (9.5, 196.25, 40) mm, rotated rx -180 ry -65 rz 88.47 deg; joints [-5.172, 14.038, -3.127, -63.862, 94.548, -64.794, -1338.473]
  MoveL 661 to (15.19, 197.47, 50) mm, rotated rx 180 ry -65 rz 93.65 deg; joints [-4.896, 13.237, -1.537, -63.743, 94.443, -63.965, -1343.653]
  MoveL 662 to (21, 199.35, 60) mm, rotated rx 180 ry -65 rz 99.09 deg; joints [-4.621, 12.299, 0.325, -63.613, 94.275, -63.014, -1349.094]
  MoveL 663 to (26.8, 201.92, 70) mm, rotated rx -180 ry -65 rz 104.77 deg; joints [-4.346, 11.124, 2.66, -63.466, 93.997, -61.853, -1354.769]
  MoveL 664 to (32.46, 205.23, 80) mm, rotated rx 180 ry -65 rz 110.65 deg; joints [-4.072, 9.32, 6.264, -63.284, 93.427, -60.121, -1360.653]
  MoveL 665 to (36.26, 208.99, 89.54) mm, rotated rx 180 ry -65 rz 116.72 deg; joints [-3.798, 7.435, 10.028, -63.109, 92.814, -58.324, -1366.718]
  MoveL 666 to (38.89, 212.87, 98.8) mm, rotated rx -180 ry -65 rz 122.94 deg; joints [-3.525, 7.41, 10.028, -63.022, 93.058, -58.228, -1372.941]
